LIN {X 0,Y 474.701,Z 198.658,A -85,B 0,C 180,E1 -7391.962,E2 -7391.962} C_VEL
LIN {X 0,Y 474.697,Z 198.664,A -85,B 0,C 180,E1 -7395.456,E2 -7395.456} C_VEL
LIN {X 0,Y 474.662,Z 198.657,A -85,B 0,C 180,E1 -7399.01,E2 -7399.01} C_VEL
LIN {X 0,Y 474.586,Z 198.681,A -85,B 0,C 180,E1 -7401.729,E2 -7401.729} C_VEL
LIN {X 0,Y 474.656,Z 198.662,A -85,B 0,C 180,E1 -7404.493,E2 -7404.493} C_VEL
LIN {X 0,Y 474.697,Z 198.662,A -85,B 0,C 180,E1 -7407.339,E2 -7407.339} C_VEL
LIN {X 0,Y 474.606,Z 198.671,A -85,B 0,C 180,E1 -7410.811,E2 -7410.811} C_VEL
LIN {X 0,Y 474.636,Z 198.675,A -85,B 0,C 180,E1 -7413.984,E2 -7413.984} C_VEL
LIN {X 0,Y 474.572,Z 198.677,A -85,B 0,C 180,E1 -7416.9,E2 -7416.9} C_VEL
LIN {X 0,Y 474.625,Z 198.675,A -85,B 0,C 180,E1 -7419.648,E2 -7419.648} C_VEL
LIN {X 0,Y 474.612,Z 198.673,A -85,B 0,C 180,E1 -7422.934,E2 -7422.934} C_VEL
LIN {X 0,Y 474.604,Z 198.679,A -85,B 0,C 180,E1 -7425.895,E2 -7425.895} C_VEL
LIN {X 0,Y 474.625,Z 198.671,A -85,B 0,C 180,E1 -7429.041,E2 -7429.041} C_VEL
LIN {X 0,Y 474.608,Z 198.678,A -85,B 0,C 180,E1 -7431.704,E2 -7431.704} C_VEL
LIN {X 0,Y 474.623,Z 198.668,A -85,B 0,C 180,E1 -7434.726,E2 -7434.726} C_VEL
LIN {X 0,Y 474.635,Z 198.669,A -85,B 0,C 180,E1 -7437.788,E2 -7437.788} C_VEL
LIN {X 0,Y 474.623,Z 198.677,A -85,B 0,C 180,E1 -7440.885,E2 -7440.885} C_VEL
LIN {X 0,Y 474.66,Z 198.672,A -85,B 0,C 180,E1 -7443.628,E2 -7443.628} C_VEL
LIN {X 0,Y 474.635,Z 198.669,A -85,B 0,C 180,E1 -7446.641,E2 -7446.641} C_VEL
LIN {X 0,Y 474.653,Z 198.661,A -85,B 0,C 180,E1 -7450.09,E2 -7450.09} C_VEL
LIN {X 0,Y 474.646,Z 198.663,A -85,B 0,C 180,E1 -7451.677,E2 -7451.677} C_VEL
LIN {X 0,Y 473.979,Z 198.754,A -85,B 0,C 180,E1 -7452.386,E2 -7452.386} C_VEL
LIN {X 0,Y 471.131,Z 199.113,A -85,B 0,C 180,E1 -7453.537,E2 -7453.537} C_VEL
LIN {X 0,Y 468.721,Z 199.413,A -85,B 0,C 180,E1 -7454.466,E2 -7454.466} C_VEL
LIN {X 0,Y 467.682,Z 199.532,A -85,B 0,C 180,E1 -7455.183,E2 -7455.183} C_VEL
LIN {X 0,Y 467.596,Z 199.539,A -85,B 0,C 180,E1 -7455.426,E2 -7455.426} C_VEL
LIN {X 0,Y 467.653,Z 199.547,A -85,B 0,C 180,E1 -7458.734,E2 -7458.734} C_VEL
LIN {X 0,Y 467.681,Z 199.542,A -85,B 0,C 180,E1 -7461.357,E2 -7461.357} C_VEL
LIN {X 0,Y 467.723,Z 199.527,A -85,B 0,C 180,E1 -7463.962,E2 -7463.962} C_VEL
LIN {X 0,Y 467.656,Z 199.646,A -85,B 0,C 180,E1 -7465.367,E2 -7465.367} C_VEL
LIN {X 0,Y 470.553,Z 208.926,A -85,B 0,C 180,E1 -7466.72,E2 -7466.72} C_VEL
LIN {X 0,Y 480.237,Z 229.746,A -85,B 0,C 180,E1 -7467.714,E2 -7467.714} C_VEL
LIN {X 0,Y 477.501,Z 414.726,A -85,B 0,C 180,E1 -7470.658,E2 -7470.658} C_VEL
LIN {X 0,Y 476.956,Z 430.924,A -85,B 0,C 180,E1 -7471.082,E2 -7471.082} C_VEL
LIN {X 0,Y 476.243,Z 446.299,A -85,B 0,C 180,E1 -7471.638,E2 -7471.638} C_VEL
LIN {X 0,Y 475.447,Z 461.115,A -85,B 0,C 180,E1 -7472.329,E2 -7472.329} C_VEL
LIN {X 0,Y 474.447,Z 475.812,A -85,B 0,C 180,E1 -7473.184,E2 -7473.184} C_VEL
LIN {X 0,Y 473.458,Z 489.457,A -85,B 0,C 180,E1 -7474.15,E2 -7474.15} C_VEL
LIN {X 0,Y 472.422,Z 503.502,A -85,B 0,C 180,E1 -7475.335,E2 -7475.335} C_VEL
LIN {X 0,Y 471.27,Z 516.574,A -85,B 0,C 180,E1 -7476.636,E2 -7476.636} C_VEL
LIN {X 0,Y 470.217,Z 529.445,A -85,B 0,C 180,E1 -7478.163,E2 -7478.163} C_VEL
LIN {X 0,Y 469.318,Z 540.358,A -85,B 0,C 180,E1 -7479.698,E2 -7479.698} C_VEL
LIN {X 0,Y 468.563,Z 549.76,A -85,B 0,C 180,E1 -7481.244,E2 -7481.244} C_VEL
LIN {X 0,Y 467.904,Z 558.942,A -85,B 0,C 180,E1 -7483.02,E2 -7483.02} C_VEL
LIN {X 0,Y 467.402,Z 566.666,A -85,B 0,C 180,E1 -7484.81,E2 -7484.81} C_VEL
LIN {X 0,Y 467.041,Z 572.995,A -85,B 0,C 180,E1 -7486.613,E2 -7486.613} C_VEL
LIN {X 0,Y 466.832,Z 578.273,A -85,B 0,C 180,E1 -7488.479,E2 -7488.479} C_VEL
LIN {X 0,Y 466.666,Z 582.208,A -85,B 0,C 180,E1 -7490.266,E2 -7490.266} C_VEL
LIN {X 0,Y 466.519,Z 585.068,A -85,B 0,C 180,E1 -7492.124,E2 -7492.124} C_VEL
LIN {X 0,Y 466.463,Z 586.873,A -85,B 0,C 180,E1 -7494.003,E2 -7494.003} C_VEL
LIN {X 0,Y 466.465,Z 587.555,A -85,B 0,C 180,E1 -7495.907,E2 -7495.907} C_VEL
LIN {X 0,Y 466.492,Z 587.024,A -85,B 0,C 180,E1 -7497.841,E2 -7497.841} C_VEL
LIN {X 0,Y 466.581,Z 585.307,A -85,B 0,C 180,E1 -7499.806,E2 -7499.806} C_VEL
LIN {X 0,Y 466.679,Z 582.29,A -85,B 0,C 180,E1 -7501.808,E2 -7501.808} C_VEL
LIN {X 0,Y 466.876,Z 577.769,A -85,B 0,C 180,E1 -7503.846,E2 -7503.846} C_VEL
LIN {X 0,Y 467.13,Z 572.464,A -85,B 0,C 180,E1 -7505.666,E2 -7505.666} C_VEL
LIN {X 0,Y 467.494,Z 565.604,A -85,B 0,C 180,E1 -7507.565,E2 -7507.565} C_VEL
LIN {X 0,Y 467.974,Z 557.8,A -85,B 0,C 180,E1 -7509.346,E2 -7509.346} C_VEL
LIN {X 0,Y 468.743,Z 547.515,A -85,B 0,C 180,E1 -7511.276,E2 -7511.276} C_VEL
LIN {X 0,Y 469.535,Z 537.645,A -85,B 0,C 180,E1 -7512.825,E2 -7512.825} C_VEL
LIN {X 0,Y 470.512,Z 526.433,A -85,B 0,C 180,E1 -7514.331,E2 -7514.331} C_VEL
LIN {X 0,Y 471.498,Z 514.718,A -85,B 0,C 180,E1 -7515.681,E2 -7515.681} C_VEL
LIN {X 0,Y 472.653,Z 500.994,A -85,B 0,C 180,E1 -7517.02,E2 -7517.02} C_VEL
LIN {X 0,Y 473.89,Z 485.591,A -85,B 0,C 180,E1 -7518.264,E2 -7518.264} C_VEL
LIN {X 0,Y 474.951,Z 470.284,A -85,B 0,C 180,E1 -7519.276,E2 -7519.276} C_VEL
LIN {X 0,Y 475.877,Z 454.74,A -85,B 0,C 180,E1 -7520.105,E2 -7520.105} C_VEL
LIN {X 0,Y 476.698,Z 438.378,A -85,B 0,C 180,E1 -7520.786,E2 -7520.786} C_VEL
LIN {X 0,Y 477.348,Z 421.885,A -85,B 0,C 180,E1 -7521.289,E2 -7521.289} C_VEL
LIN {X 0,Y 477.799,Z 404.177,A -85,B 0,C 180,E1 -7521.642,E2 -7521.642} C_VEL
LIN {X 0,Y 480.393,Z 230.17,A -85,B 0,C 180,E1 -7524.41,E2 -7524.41} C_VEL
LIN {X 0,Y 471.537,Z 211.431,A -85,B 0,C 180,E1 -7525.341,E2 -7525.341} C_VEL
LIN {X 0,Y 470.535,Z 209.235,A -85,B 0,C 180,E1 -7525.46,E2 -7525.46} C_VEL
LIN {X 0,Y 467.562,Z 199.56,A -85,B 0,C 180,E1 -7526.952,E2 -7526.952} C_VEL
LIN {X 0,Y 467.56,Z 199.557,A -85,B 0,C 180,E1 -7529.266,E2 -7529.266} C_VEL
LIN {X 0,Y 467.596,Z 199.554,A -85,B 0,C 180,E1 -7532.469,E2 -7532.469} C_VEL
LIN {X 0,Y 467.552,Z 199.556,A -85,B 0,C 180,E1 -7535.11,E2 -7535.11} C_VEL
LIN {X 0,Y 467.526,Z 199.554,A -85,B 0,C 180,E1 -7537.926,E2 -7537.926} C_VEL
LIN {X 0,Y 467.615,Z 199.547,A -85,B 0,C 180,E1 -7540.692,E2 -7540.692} C_VEL
LIN {X 0,Y 467.642,Z 199.541,A -85,B 0,C 180,E1 -7544.115,E2 -7544.115} C_VEL
LIN {X 0,Y 467.647,Z 199.538,A -85,B 0,C 180,E1 -7547.642,E2 -7547.642} C_VEL
LIN {X 0,Y 467.654,Z 199.547,A -85,B 0,C 180,E1 -7550.485,E2 -7550.485} C_VEL
LIN {X 0,Y 467.683,Z 199.537,A -85,B 0,C 180,E1 -7553.095,E2 -7553.095} C_VEL
LIN {X 0,Y 467.712,Z 199.536,A -85,B 0,C 180,E1 -7554.827,E2 -7554.827} C_VEL
LIN {X 0,Y 467.851,Z 199.517,A -85,B 0,C 180,E1 -7557.417,E2 -7557.417} C_VEL
LIN {X 0,Y 467.875,Z 199.518,A -85,B 0,C 180,E1 -7560,E2 -7560} C_VEL
LIN {X 0,Y 467.852,Z 199.518,A -85,B 0,C 180,E1 -7562.583,E2 -7562.583} C_VEL
LIN {X 0,Y 467.736,Z 199.534,A -85,B 0,C 180,E1 -7566.037,E2 -7566.037} C_VEL
LIN {X 0,Y 467.675,Z 199.54,A -85,B 0,C 180,E1 -7568.643,E2 -7568.643} C_VEL
LIN {X 0,Y 467.649,Z 199.548,A -85,B 0,C 180,E1 -7572.146,E2 -7572.146} C_VEL
LIN {X 0,Y 467.632,Z 199.549,A -85,B 0,C 180,E1 -7575.695,E2 -7575.695} C_VEL
LIN {X 0,Y 467.611,Z 199.545,A -85,B 0,C 180,E1 -7578.765,E2 -7578.765} C_VEL
LIN {X 0,Y 467.574,Z 199.554,A -85,B 0,C 180,E1 -7581.269,E2 -7581.269} C_VEL
LIN {X 0,Y 467.567,Z 199.555,A -85,B 0,C 180,E1 -7583.943,E2 -7583.943} C_VEL
LIN {X 0,Y 467.621,Z 199.544,A -85,B 0,C 180,E1 -7586.8,E2 -7586.8} C_VEL
LIN {X 0,Y 467.548,Z 199.561,A -85,B 0,C 180,E1 -7589.738,E2 -7589.738} C_VEL
LIN {X 0,Y 467.578,Z 199.554,A -85,B 0,C 180,E1 -7592.759,E2 -7592.759} C_VEL
LIN {X 0,Y 467.548,Z 199.559,A -85,B 0,C 180,E1 -7595.89,E2 -7595.89} C_VEL
LIN {X 0,Y 467.577,Z 199.56,A -85,B 0,C 180,E1 -7599.145,E2 -7599.145} C_VEL
LIN {X 0,Y 467.581,Z 199.555,A -85,B 0,C 180,E1 -7602.567,E2 -7602.567} C_VEL
LIN {X 0,Y 467.565,Z 199.562,A -85,B 0,C 180,E1 -7605.054,E2 -7605.054} C_VEL
LIN {X 0,Y 467.584,Z 199.557,A -85,B 0,C 180,E1 -7607.44,E2 -7607.44} C_VEL
LIN {X 0,Y 467.578,Z 199.556,A -85,B 0,C 180,E1 -7610.856,E2 -7610.856} C_VEL
LIN {X 0,Y 467.555,Z 199.558,A -85,B 0,C 180,E1 -7614.261,E2 -7614.261} C_VEL
LIN {X 0,Y 467.623,Z 199.676,A -85,B 0,C 180,E1 -7616.717,E2 -7616.717} C_VEL
LIN {X 0,Y 473.655,Z 219.02,A -85,B 0,C 180,E1 -7619.383,E2 -7619.383} C_VEL
LIN {X 0,Y 475.73,Z 226.359,A -85,B 0,C 180,E1 -7620.338,E2 -7620.338} C_VEL
LIN {X 0,Y 475.601,Z 231.753,A -85,B 0,C 180,E1 -7620.923,E2 -7620.923} C_VEL
LIN {X 0,Y 480.058,Z 257.266,A -85,B 0,C 180,E1 -7621.669,E2 -7621.669} C_VEL
LIN {X 0,Y 478.155,Z 385.84,A -85,B 0,C 180,E1 -7623.713,E2 -7623.713} C_VEL
LIN {X 0,Y 477.384,Z 438.968,A -85,B 0,C 180,E1 -7624.572,E2 -7624.572} C_VEL
LIN {X 0,Y 476.72,Z 455.187,A -85,B 0,C 180,E1 -7624.981,E2 -7624.981} C_VEL
LIN {X 0,Y 475.931,Z 471.769,A -85,B 0,C 180,E1 -7625.577,E2 -7625.577} C_VEL
LIN {X 0,Y 475.084,Z 485.876,A -85,B 0,C 180,E1 -7626.228,E2 -7626.228} C_VEL
LIN {X 0,Y 474.059,Z 501.348,A -85,B 0,C 180,E1 -7627.124,E2 -7627.124} C_VEL
LIN {X 0,Y 472.982,Z 514.94,A -85,B 0,C 180,E1 -7628.079,E2 -7628.079} C_VEL
LIN {X 0,Y 471.805,Z 529.315,A -85,B 0,C 180,E1 -7629.282,E2 -7629.282} C_VEL
LIN {X 0,Y 470.709,Z 542.794,A -85,B 0,C 180,E1 -7630.625,E2 -7630.625} C_VEL
LIN {X 0,Y 469.852,Z 553.86,A -85,B 0,C 180,E1 -7631.919,E2 -7631.919} C_VEL
LIN {X 0,Y 468.922,Z 565.152,A -85,B 0,C 180,E1 -7633.456,E2 -7633.456} C_VEL
LIN {X 0,Y 468.276,Z 574.848,A -85,B 0,C 180,E1 -7634.996,E2 -7634.996} C_VEL
LIN {X 0,Y 467.651,Z 584.267,A -85,B 0,C 180,E1 -7636.752,E2 -7636.752} C_VEL
LIN {X 0,Y 467.337,Z 591.16,A -85,B 0,C 180,E1 -7638.287,E2 -7638.287} C_VEL
LIN {X 0,Y 466.969,Z 597.843,A -85,B 0,C 180,E1 -7640.034,E2 -7640.034} C_VEL
LIN {X 0,Y 466.79,Z 603.262,A -85,B 0,C 180,E1 -7641.777,E2 -7641.777} C_VEL
LIN {X 0,Y 466.748,Z 607.738,A -85,B 0,C 180,E1 -7643.607,E2 -7643.607} C_VEL
LIN {X 0,Y 466.599,Z 611.426,A -85,B 0,C 180,E1 -7645.681,E2 -7645.681} C_VEL
LIN {X 0,Y 466.651,Z 613.384,A -85,B 0,C 180,E1 -7647.411,E2 -7647.411} C_VEL
LIN {X 0,Y 466.615,Z 614.358,A -85,B 0,C 180,E1 -7649.137,E2 -7649.137} C_VEL
LIN {X 0,Y 466.615,Z 614.364,A -85,B 0,C 180,E1 -7650.863,E2 -7650.863} C_VEL
LIN {X 0,Y 466.651,Z 613.402,A -85,B 0,C 180,E1 -7652.59,E2 -7652.59} C_VEL
LIN {X 0,Y 466.599,Z 611.458,A -85,B 0,C 180,E1 -7654.319,E2 -7654.319} C_VEL
LIN {X 0,Y 466.749,Z 607.791,A -85,B 0,C 180,E1 -7656.393,E2 -7656.393} C_VEL
LIN {X 0,Y 466.791,Z 603.33,A -85,B 0,C 180,E1 -7658.223,E2 -7658.223} C_VEL
LIN {X 0,Y 466.97,Z 597.926,A -85,B 0,C 180,E1 -7659.967,E2 -7659.967} C_VEL
LIN {X 0,Y 467.341,Z 591.258,A -85,B 0,C 180,E1 -7661.714,E2 -7661.714} C_VEL
LIN {X 0,Y 467.737,Z 583.265,A -85,B 0,C 180,E1 -7663.468,E2 -7663.468} C_VEL
LIN {X 0,Y 468.437,Z 573.726,A -85,B 0,C 180,E1 -7665.222,E2 -7665.222} C_VEL
LIN {X 0,Y 469.225,Z 562.294,A -85,B 0,C 180,E1 -7666.982,E2 -7666.982} C_VEL
LIN {X 0,Y 470.17,Z 550.41,A -85,B 0,C 180,E1 -7668.52,E2 -7668.52} C_VEL
LIN {X 0,Y 471.132,Z 538.262,A -85,B 0,C 180,E1 -7669.864,E2 -7669.864} C_VEL
LIN {X 0,Y 472.226,Z 524.526,A -85,B 0,C 180,E1 -7671.156,E2 -7671.156} C_VEL
LIN {X 0,Y 473.297,Z 510.729,A -85,B 0,C 180,E1 -7672.25,E2 -7672.25} C_VEL
LIN {X 0,Y 474.486,Z 494.972,A -85,B 0,C 180,E1 -7673.273,E2 -7673.273} C_VEL
LIN {X 0,Y 475.503,Z 479.167,A -85,B 0,C 180,E1 -7674.098,E2 -7674.098} C_VEL
LIN {X 0,Y 476.37,Z 463.217,A -85,B 0,C 180,E1 -7674.748,E2 -7674.748} C_VEL
LIN {X 0,Y 477.018,Z 447.128,A -85,B 0,C 180,E1 -7675.236,E2 -7675.236} C_VEL
LIN {X 0,Y 477.593,Z 430.192,A -85,B 0,C 180,E1 -7675.571,E2 -7675.571} C_VEL
LIN {X 0,Y 479.963,Z 257.006,A -85,B 0,C 180,E1 -7678.31,E2 -7678.31} C_VEL
LIN {X 0,Y 475.587,Z 232.12,A -85,B 0,C 180,E1 -7679.04,E2 -7679.04} C_VEL
LIN {X 0,Y 475.709,Z 226.306,A -85,B 0,C 180,E1 -7679.667,E2 -7679.667} C_VEL
LIN {X 0,Y 470.359,Z 208.522,A -85,B 0,C 180,E1 -7682.012,E2 -7682.012} C_VEL
LIN {X 0,Y 467.612,Z 199.535,A -85,B 0,C 180,E1 -7683.269,E2 -7683.269} C_VEL
LIN {X 0,Y 467.549,Z 199.558,A -85,B 0,C 180,E1 -7685.89,E2 -7685.89} C_VEL
LIN {X 0,Y 467.568,Z 199.557,A -85,B 0,C 180,E1 -7689.146,E2 -7689.146} C_VEL
LIN {X 0,Y 467.57,Z 199.557,A -85,B 0,C 180,E1 -7691.403,E2 -7691.403} C_VEL
LIN {X 0,Y 467.562,Z 199.554,A -85,B 0,C 180,E1 -7695.052,E2 -7695.052} C_VEL
LIN {X 0,Y 467.57,Z 199.555,A -85,B 0,C 180,E1 -7698.597,E2 -7698.597} C_VEL
LIN {X 0,Y 467.561,Z 199.554,A -85,B 0,C 180,E1 -7701.955,E2 -7701.955} C_VEL
LIN {X 0,Y 467.555,Z 199.558,A -85,B 0,C 180,E1 -7705.167,E2 -7705.167} C_VEL
LIN {X 0,Y 467.579,Z 199.545,A -85,B 0,C 180,E1 -7708.26,E2 -7708.26} C_VEL
LIN {X 0,Y 467.572,Z 199.554,A -85,B 0,C 180,E1 -7711.25,E2 -7711.25} C_VEL
LIN {X 0,Y 467.594,Z 199.539,A -85,B 0,C 180,E1 -7714.159,E2 -7714.159} C_VEL
LIN {X 0,Y 467.572,Z 199.556,A -85,B 0,C 180,E1 -7716.996,E2 -7716.996} C_VEL
LIN {X 0,Y 467.618,Z 199.539,A -85,B 0,C 180,E1 -7719.777,E2 -7719.777} C_VEL
LIN {X 0,Y 467.592,Z 199.546,A -85,B 0,C 180,E1 -7722.506,E2 -7722.506} C_VEL
LIN {X 0,Y 467.602,Z 199.547,A -85,B 0,C 180,E1 -7725.196,E2 -7725.196} C_VEL
LIN {X 0,Y 467.653,Z 199.53,A -85,B 0,C 180,E1 -7727.855,E2 -7727.855} C_VEL
LIN {X 0,Y 467.667,Z 199.538,A -85,B 0,C 180,E1 -7731.357,E2 -7731.357} C_VEL
LIN {X 0,Y 467.73,Z 199.534,A -85,B 0,C 180,E1 -7733.962,E2 -7733.962} C_VEL
LIN {X 0,Y 467.854,Z 199.495,A -85,B 0,C 180,E1 -7737.417,E2 -7737.417} C_VEL
LIN {X 0,Y 467.878,Z 199.511,A -85,B 0,C 180,E1 -7740,E2 -7740} C_VEL
LIN {X 0,Y 467.855,Z 199.517,A -85,B 0,C 180,E1 -7742.583,E2 -7742.583} C_VEL
LIN {X 0,Y 467.739,Z 199.524,A -85,B 0,C 180,E1 -7746.037,E2 -7746.037} C_VEL
LIN {X 0,Y 467.677,Z 199.539,A -85,B 0,C 180,E1 -7748.643,E2 -7748.643} C_VEL
LIN {X 0,Y 467.653,Z 199.535,A -85,B 0,C 180,E1 -7752.145,E2 -7752.145} C_VEL
LIN {X 0,Y 467.636,Z 199.546,A -85,B 0,C 180,E1 -7755.695,E2 -7755.695} C_VEL
LIN {X 0,Y 467.614,Z 199.534,A -85,B 0,C 180,E1 -7758.765,E2 -7758.765} C_VEL
LIN {X 0,Y 467.578,Z 199.549,A -85,B 0,C 180,E1 -7761.268,E2 -7761.268} C_VEL
LIN {X 0,Y 467.571,Z 199.55,A -85,B 0,C 180,E1 -7763.943,E2 -7763.943} C_VEL
LIN {X 0,Y 467.614,Z 199.541,A -85,B 0,C 180,E1 -7766.8,E2 -7766.8} C_VEL
LIN {X 0,Y 467.584,Z 199.555,A -85,B 0,C 180,E1 -7769.736,E2 -7769.736} C_VEL
LIN {X 0,Y 467.581,Z 199.543,A -85,B 0,C 180,E1 -7772.758,E2 -7772.758} C_VEL
LIN {X 0,Y 467.554,Z 199.556,A -85,B 0,C 180,E1 -7775.889,E2 -7775.889} C_VEL
LIN {X 0,Y 467.579,Z 199.545,A -85,B 0,C 180,E1 -7779.145,E2 -7779.145} C_VEL
LIN {X 0,Y 467.584,Z 199.547,A -85,B 0,C 180,E1 -7782.567,E2 -7782.567} C_VEL
LIN {X 0,Y 467.563,Z 199.55,A -85,B 0,C 180,E1 -7785.053,E2 -7785.053} C_VEL
LIN {X 0,Y 467.587,Z 199.554,A -85,B 0,C 180,E1 -7787.44,E2 -7787.44} C_VEL
LIN {X 0,Y 467.558,Z 199.553,A -85,B 0,C 180,E1 -7790.853,E2 -7790.853} C_VEL
LIN {X 0,Y 467.558,Z 199.547,A -85,B 0,C 180,E1 -7794.261,E2 -7794.261} C_VEL
LIN {X 0,Y 467.581,Z 199.554,A -85,B 0,C 180,E1 -7797.321,E2 -7797.321} C_VEL
LIN {X 0,Y 467.569,Z 199.554,A -85,B 0,C 180,E1 -7800.667,E2 -7800.667} C_VEL
LIN {X 0,Y 467.616,Z 199.547,A -85,B 0,C 180,E1 -7803.2,E2 -7803.2} C_VEL
LIN {X 0,Y 467.592,Z 199.545,A -85,B 0,C 180,E1 -7806.468,E2 -7806.468} C_VEL
LIN {X 0,Y 467.622,Z 199.538,A -85,B 0,C 180,E1 -7809.777,E2 -7809.777} C_VEL
LIN {X 0,Y 467.597,Z 199.545,A -85,B 0,C 180,E1 -7812.506,E2 -7812.506} C_VEL
LIN {X 0,Y 467.605,Z 199.541,A -85,B 0,C 180,E1 -7815.196,E2 -7815.196} C_VEL
LIN {X 0,Y 467.596,Z 199.539,A -85,B 0,C 180,E1 -7815.426,E2 -7815.426} C_VEL
LIN {X 0,Y 466.926,Z 199.621,A -85,B 0,C 180,E1 -7816.145,E2 -7816.145} C_VEL
LIN {X 0,Y 464.083,Z 199.985,A -85,B 0,C 180,E1 -7817.314,E2 -7817.314} C_VEL
LIN {X 0,Y 461.684,Z 200.288,A -85,B 0,C 180,E1 -7818.256,E2 -7818.256} C_VEL
LIN {X 0,Y 460.658,Z 200.416,A -85,B 0,C 180,E1 -7818.983,E2 -7818.983} C_VEL
LIN {X 0,Y 460.576,Z 200.425,A -85,B 0,C 180,E1 -7819.23,E2 -7819.23} C_VEL
LIN {X 0,Y 460.669,Z 200.411,A -85,B 0,C 180,E1 -7822.587,E2 -7822.587} C_VEL
LIN {X 0,Y 460.655,Z 200.475,A -85,B 0,C 180,E1 -7824.94,E2 -7824.94} C_VEL
LIN {X 0,Y 463.309,Z 209.246,A -85,B 0,C 180,E1 -7826.227,E2 -7826.227} C_VEL
LIN {X 0,Y 470.395,Z 224.099,A -85,B 0,C 180,E1 -7826.973,E2 -7826.973} C_VEL
LIN {X 0,Y 473.966,Z 231.809,A -85,B 0,C 180,E1 -7827.344,E2 -7827.344} C_VEL
LIN {X 0,Y 471.072,Z 414.547,A -85,B 0,C 180,E1 -7830.288,E2 -7830.288} C_VEL
LIN {X 0,Y 470.511,Z 430.619,A -85,B 0,C 180,E1 -7830.708,E2 -7830.708} C_VEL
LIN {X 0,Y 469.744,Z 446.47,A -85,B 0,C 180,E1 -7831.286,E2 -7831.286} C_VEL
LIN {X 0,Y 468.982,Z 460.305,A -85,B 0,C 180,E1 -7831.932,E2 -7831.932} C_VEL
LIN {X 0,Y 467.809,Z 476.864,A -85,B 0,C 180,E1 -7832.906,E2 -7832.906} C_VEL
LIN {X 0,Y 466.677,Z 491.742,A -85,B 0,C 180,E1 -7833.994,E2 -7833.994} C_VEL
LIN {X 0,Y 465.566,Z 505.446,A -85,B 0,C 180,E1 -7835.196,E2 -7835.196} C_VEL
LIN {X 0,Y 464.375,Z 518.236,A -85,B 0,C 180,E1 -7836.517,E2 -7836.517} C_VEL
LIN {X 0,Y 463.266,Z 530.89,A -85,B 0,C 180,E1 -7838.066,E2 -7838.066} C_VEL
LIN {X 0,Y 462.337,Z 541.697,A -85,B 0,C 180,E1 -7839.625,E2 -7839.625} C_VEL
LIN {X 0,Y 461.458,Z 552.148,A -85,B 0,C 180,E1 -7841.419,E2 -7841.419} C_VEL
LIN {X 0,Y 460.771,Z 560.953,A -85,B 0,C 180,E1 -7843.225,E2 -7843.225} C_VEL
LIN {X 0,Y 460.282,Z 568.34,A -85,B 0,C 180,E1 -7845.044,E2 -7845.044} C_VEL
LIN {X 0,Y 459.953,Z 574.477,A -85,B 0,C 180,E1 -7846.876,E2 -7846.876} C_VEL
LIN {X 0,Y 459.733,Z 579.339,A -85,B 0,C 180,E1 -7848.725,E2 -7848.725} C_VEL
LIN {X 0,Y 459.539,Z 583.111,A -85,B 0,C 180,E1 -7850.594,E2 -7850.594} C_VEL
LIN {X 0,Y 459.405,Z 585.806,A -85,B 0,C 180,E1 -7852.485,E2 -7852.485} C_VEL
LIN {X 0,Y 459.364,Z 587.309,A -85,B 0,C 180,E1 -7854.398,E2 -7854.398} C_VEL
LIN {X 0,Y 459.377,Z 587.734,A -85,B 0,C 180,E1 -7856.338,E2 -7856.338} C_VEL
LIN {X 0,Y 459.411,Z 586.996,A -85,B 0,C 180,E1 -7858.309,E2 -7858.309} C_VEL
LIN {X 0,Y 459.494,Z 584.949,A -85,B 0,C 180,E1 -7860.313,E2 -7860.313} C_VEL
LIN {X 0,Y 459.646,Z 581.583,A -85,B 0,C 180,E1 -7862.353,E2 -7862.353} C_VEL
LIN {X 0,Y 459.884,Z 576.747,A -85,B 0,C 180,E1 -7864.432,E2 -7864.432} C_VEL
LIN {X 0,Y 460.141,Z 571.404,A -85,B 0,C 180,E1 -7866.215,E2 -7866.215} C_VEL
LIN {X 0,Y 460.574,Z 564.098,A -85,B 0,C 180,E1 -7868.169,E2 -7868.169} C_VEL
LIN {X 0,Y 461.206,Z 555.292,A -85,B 0,C 180,E1 -7870.096,E2 -7870.096} C_VEL
LIN {X 0,Y 461.998,Z 545.931,A -85,B 0,C 180,E1 -7871.807,E2 -7871.807} C_VEL
LIN {X 0,Y 462.872,Z 535.742,A -85,B 0,C 180,E1 -7873.395,E2 -7873.395} C_VEL
LIN {X 0,Y 463.949,Z 524.199,A -85,B 0,C 180,E1 -7874.916,E2 -7874.916} C_VEL
LIN {X 0,Y 465.058,Z 511.855,A -85,B 0,C 180,E1 -7876.298,E2 -7876.298} C_VEL
LIN {X 0,Y 466.213,Z 497.981,A -85,B 0,C 180,E1 -7877.616,E2 -7877.616} C_VEL
LIN {X 0,Y 467.414,Z 483.724,A -85,B 0,C 180,E1 -7878.745,E2 -7878.745} C_VEL
LIN {X 0,Y 468.469,Z 469.786,A -85,B 0,C 180,E1 -7879.665,E2 -7879.665} C_VEL
LIN {X 0,Y 469.488,Z 453.715,A -85,B 0,C 180,E1 -7880.52,E2 -7880.52} C_VEL
LIN {X 0,Y 470.295,Z 437.805,A -85,B 0,C 180,E1 -7881.179,E2 -7881.179} C_VEL
LIN {X 0,Y 471.011,Z 421.355,A -85,B 0,C 180,E1 -7881.675,E2 -7881.675} C_VEL
LIN {X 0,Y 471.426,Z 404.144,A -85,B 0,C 180,E1 -7882.021,E2 -7882.021} C_VEL
LIN {X 0,Y 474.192,Z 232.29,A -85,B 0,C 180,E1 -7884.79,E2 -7884.79} C_VEL
LIN {X 0,Y 464.605,Z 212.097,A -85,B 0,C 180,E1 -7885.828,E2 -7885.828} C_VEL
LIN {X 0,Y 463.367,Z 209.366,A -85,B 0,C 180,E1 -7885.993,E2 -7885.993} C_VEL
LIN {X 0,Y 460.528,Z 200.433,A -85,B 0,C 180,E1 -7887.397,E2 -7887.397} C_VEL
LIN {X 0,Y 460.519,Z 200.434,A -85,B 0,C 180,E1 -7890.768,E2 -7890.768} C_VEL
LIN {X 0,Y 460.511,Z 200.434,A -85,B 0,C 180,E1 -7893.732,E2 -7893.732} C_VEL
LIN {X 0,Y 460.536,Z 200.434,A -85,B 0,C 180,E1 -7896.624,E2 -7896.624} C_VEL
LIN {X 0,Y 460.543,Z 200.431,A -85,B 0,C 180,E1 -7899.452,E2 -7899.452} C_VEL
LIN {X 0,Y 460.542,Z 200.43,A -85,B 0,C 180,E1 -7902.23,E2 -7902.23} C_VEL
LIN {X 0,Y 460.557,Z 200.426,A -85,B 0,C 180,E1 -7904.965,E2 -7904.965} C_VEL
LIN {X 0,Y 460.603,Z 200.417,A -85,B 0,C 180,E1 -7908.559,E2 -7908.559} C_VEL
LIN {X 0,Y 460.613,Z 200.419,A -85,B 0,C 180,E1 -7911.224,E2 -7911.224} C_VEL
LIN {X 0,Y 460.691,Z 200.408,A -85,B 0,C 180,E1 -7913.87,E2 -7913.87} C_VEL
LIN {X 0,Y 460.792,Z 200.396,A -85,B 0,C 180,E1 -7917.377,E2 -7917.377} C_VEL
LIN {X 0,Y 460.845,Z 200.394,A -85,B 0,C 180,E1 -7920,E2 -7920} C_VEL
LIN {X 0,Y 460.793,Z 200.397,A -85,B 0,C 180,E1 -7922.623,E2 -7922.623} C_VEL
LIN {X 0,Y 460.702,Z 200.411,A -85,B 0,C 180,E1 -7926.13,E2 -7926.13} C_VEL
LIN {X 0,Y 460.622,Z 200.418,A -85,B 0,C 180,E1 -7928.776,E2 -7928.776} C_VEL
LIN {X 0,Y 460.607,Z 200.422,A -85,B 0,C 180,E1 -7932.445,E2 -7932.445} C_VEL
LIN {X 0,Y 460.593,Z 200.424,A -85,B 0,C 180,E1 -7935.998,E2 -7935.998} C_VEL
LIN {X 0,Y 460.564,Z 200.423,A -85,B 0,C 180,E1 -7938.902,E2 -7938.902} C_VEL
LIN {X 0,Y 460.51,Z 200.435,A -85,B 0,C 180,E1 -7941.486,E2 -7941.486} C_VEL
LIN {X 0,Y 460.536,Z 200.428,A -85,B 0,C 180,E1 -7944.332,E2 -7944.332} C_VEL
LIN {X 0,Y 460.578,Z 200.424,A -85,B 0,C 180,E1 -7947.243,E2 -7947.243} C_VEL
LIN {X 0,Y 460.505,Z 200.434,A -85,B 0,C 180,E1 -7950.24,E2 -7950.24} C_VEL
LIN {X 0,Y 460.523,Z 200.436,A -85,B 0,C 180,E1 -7953.325,E2 -7953.325} C_VEL
LIN {X 0,Y 460.471,Z 200.439,A -85,B 0,C 180,E1 -7956.53,E2 -7956.53} C_VEL
LIN {X 0,Y 460.527,Z 200.434,A -85,B 0,C 180,E1 -7959.863,E2 -7959.863} C_VEL
LIN {X 0,Y 460.508,Z 200.44,A -85,B 0,C 180,E1 -7962.901,E2 -7962.901} C_VEL
LIN {X 0,Y 460.506,Z 200.437,A -85,B 0,C 180,E1 -7965.831,E2 -7965.831} C_VEL
LIN {X 0,Y 460.526,Z 200.435,A -85,B 0,C 180,E1 -7968.989,E2 -7968.989} C_VEL
LIN {X 0,Y 460.522,Z 200.435,A -85,B 0,C 180,E1 -7971.267,E2 -7971.267} C_VEL
LIN {X 0,Y 460.506,Z 200.437,A -85,B 0,C 180,E1 -7974.555,E2 -7974.555} C_VEL
LIN {X 0,Y 460.575,Z 200.515,A -85,B 0,C 180,E1 -7976.247,E2 -7976.247} C_VEL
LIN {X 0,Y 466.904,Z 220.645,A -85,B 0,C 180,E1 -7979.09,E2 -7979.09} C_VEL
LIN {X 0,Y 469.168,Z 228.639,A -85,B 0,C 180,E1 -7980.153,E2 -7980.153} C_VEL
LIN {X 0,Y 469.148,Z 231.612,A -85,B 0,C 180,E1 -7980.485,E2 -7980.485} C_VEL
LIN {X 0,Y 473.829,Z 258.396,A -85,B 0,C 180,E1 -7981.278,E2 -7981.278} C_VEL
LIN {X 0,Y 472.073,Z 367.989,A -85,B 0,C 180,E1 -7983.043,E2 -7983.043} C_VEL
LIN {X 0,Y 470.982,Z 439.154,A -85,B 0,C 180,E1 -7984.207,E2 -7984.207} C_VEL
LIN {X 0,Y 470.254,Z 455.927,A -85,B 0,C 180,E1 -7984.643,E2 -7984.643} C_VEL
LIN {X 0,Y 469.454,Z 471.57,A -85,B 0,C 180,E1 -7985.218,E2 -7985.218} C_VEL
LIN {X 0,Y 468.538,Z 485.67,A -85,B 0,C 180,E1 -7985.875,E2 -7985.875} C_VEL
LIN {X 0,Y 467.506,Z 500.567,A -85,B 0,C 180,E1 -7986.747,E2 -7986.747} C_VEL
LIN {X 0,Y 466.318,Z 514.722,A -85,B 0,C 180,E1 -7987.75,E2 -7987.75} C_VEL
LIN {X 0,Y 465.094,Z 529.093,A -85,B 0,C 180,E1 -7988.969,E2 -7988.969} C_VEL
LIN {X 0,Y 464.022,Z 541.237,A -85,B 0,C 180,E1 -7990.179,E2 -7990.179} C_VEL
LIN {X 0,Y 463.004,Z 553.639,A -85,B 0,C 180,E1 -7991.642,E2 -7991.642} C_VEL
LIN {X 0,Y 462.009,Z 564.929,A -85,B 0,C 180,E1 -7993.201,E2 -7993.201} C_VEL
LIN {X 0,Y 461.336,Z 574.626,A -85,B 0,C 180,E1 -7994.765,E2 -7994.765} C_VEL
LIN {X 0,Y 460.646,Z 584.047,A -85,B 0,C 180,E1 -7996.546,E2 -7996.546} C_VEL
LIN {X 0,Y 460.166,Z 592.774,A -85,B 0,C 180,E1 -7998.548,E2 -7998.548} C_VEL
LIN {X 0,Y 459.775,Z 600.512,A -85,B 0,C 180,E1 -8000.764,E2 -8000.764} C_VEL
LIN {X 0,Y 459.647,Z 606.401,A -85,B 0,C 180,E1 -8002.974,E2 -8002.974} C_VEL
LIN {X 0,Y 459.578,Z 609.849,A -85,B 0,C 180,E1 -8004.736,E2 -8004.736} C_VEL
LIN {X 0,Y 459.53,Z 612.355,A -85,B 0,C 180,E1 -8006.493,E2 -8006.493} C_VEL
LIN {X 0,Y 459.537,Z 613.773,A -85,B 0,C 180,E1 -8008.247,E2 -8008.247} C_VEL
LIN {X 0,Y 459.525,Z 614.311,A -85,B 0,C 180,E1 -8010,E2 -8010} C_VEL
LIN {X 0,Y 459.537,Z 613.787,A -85,B 0,C 180,E1 -8011.753,E2 -8011.753} C_VEL
LIN {X 0,Y 459.53,Z 612.382,A -85,B 0,C 180,E1 -8013.507,E2 -8013.507} C_VEL
LIN {X 0,Y 459.578,Z 609.892,A -85,B 0,C 180,E1 -8015.265,E2 -8015.265} C_VEL
LIN {X 0,Y 459.648,Z 606.461,A -85,B 0,C 180,E1 -8017.026,E2 -8017.026} C_VEL
LIN {X 0,Y 459.782,Z 600.591,A -85,B 0,C 180,E1 -8019.236,E2 -8019.236} C_VEL
LIN {X 0,Y 460.172,Z 592.867,A -85,B 0,C 180,E1 -8021.452,E2 -8021.452} C_VEL
LIN {X 0,Y 460.648,Z 584.155,A -85,B 0,C 180,E1 -8023.454,E2 -8023.454} C_VEL
LIN {X 0,Y 461.36,Z 574.747,A -85,B 0,C 180,E1 -8025.235,E2 -8025.235} C_VEL
LIN {X 0,Y 462.071,Z 565.053,A -85,B 0,C 180,E1 -8026.797,E2 -8026.797} C_VEL
LIN {X 0,Y 463.008,Z 553.755,A -85,B 0,C 180,E1 -8028.359,E2 -8028.359} C_VEL
LIN {X 0,Y 464.066,Z 541.342,A -85,B 0,C 180,E1 -8029.82,E2 -8029.82} C_VEL
LIN {X 0,Y 465.212,Z 527.998,A -85,B 0,C 180,E1 -8031.142,E2 -8031.142} C_VEL
LIN {X 0,Y 466.32,Z 514.76,A -85,B 0,C 180,E1 -8032.251,E2 -8032.251} C_VEL
LIN {X 0,Y 467.497,Z 500.499,A -85,B 0,C 180,E1 -8033.256,E2 -8033.256} C_VEL
LIN {X 0,Y 468.552,Z 485.569,A -85,B 0,C 180,E1 -8034.125,E2 -8034.125} C_VEL
LIN {X 0,Y 469.517,Z 470.032,A -85,B 0,C 180,E1 -8034.838,E2 -8034.838} C_VEL
LIN {X 0,Y 470.27,Z 453.573,A -85,B 0,C 180,E1 -8035.416,E2 -8035.416} C_VEL
LIN {X 0,Y 470.954,Z 436.774,A -85,B 0,C 180,E1 -8035.819,E2 -8035.819} C_VEL
LIN {X 0,Y 473.743,Z 259.378,A -85,B 0,C 180,E1 -8038.667,E2 -8038.667} C_VEL
LIN {X 0,Y 469.08,Z 232.203,A -85,B 0,C 180,E1 -8039.446,E2 -8039.446} C_VEL
LIN {X 0,Y 469.044,Z 228.304,A -85,B 0,C 180,E1 -8039.881,E2 -8039.881} C_VEL
LIN {X 0,Y 463.548,Z 209.982,A -85,B 0,C 180,E1 -8042.338,E2 -8042.338} C_VEL
LIN {X 0,Y 460.544,Z 200.421,A -85,B 0,C 180,E1 -8043.717,E2 -8043.717} C_VEL
LIN {X 0,Y 460.47,Z 200.442,A -85,B 0,C 180,E1 -8046.53,E2 -8046.53} C_VEL
LIN {X 0,Y 460.518,Z 200.428,A -85,B 0,C 180,E1 -8049.863,E2 -8049.863} C_VEL
LIN {X 0,Y 460.489,Z 200.434,A -85,B 0,C 180,E1 -8052.897,E2 -8052.897} C_VEL
LIN {X 0,Y 460.502,Z 200.428,A -85,B 0,C 180,E1 -8055.831,E2 -8055.831} C_VEL
LIN {X 0,Y 460.524,Z 200.428,A -85,B 0,C 180,E1 -8058.988,E2 -8058.988} C_VEL
LIN {X 0,Y 460.513,Z 200.436,A -85,B 0,C 180,E1 -8061.266,E2 -8061.266} C_VEL
LIN {X 0,Y 460.505,Z 200.428,A -85,B 0,C 180,E1 -8064.554,E2 -8064.554} C_VEL
LIN {X 0,Y 460.527,Z 200.423,A -85,B 0,C 180,E1 -8067.715,E2 -8067.715} C_VEL
LIN {X 0,Y 460.535,Z 200.434,A -85,B 0,C 180,E1 -8070.769,E2 -8070.769} C_VEL
LIN {X 0,Y 460.552,Z 200.415,A -85,B 0,C 180,E1 -8073.734,E2 -8073.734} C_VEL
LIN {X 0,Y 460.541,Z 200.432,A -85,B 0,C 180,E1 -8076.624,E2 -8076.624} C_VEL
LIN {X 0,Y 460.547,Z 200.419,A -85,B 0,C 180,E1 -8079.453,E2 -8079.453} C_VEL
LIN {X 0,Y 460.544,Z 200.42,A -85,B 0,C 180,E1 -8082.23,E2 -8082.23} C_VEL
LIN {X 0,Y 460.561,Z 200.426,A -85,B 0,C 180,E1 -8084.965,E2 -8084.965} C_VEL
LIN {X 0,Y 460.607,Z 200.405,A -85,B 0,C 180,E1 -8088.559,E2 -8088.559} C_VEL
LIN {X 0,Y 460.617,Z 200.416,A -85,B 0,C 180,E1 -8091.224,E2 -8091.224} C_VEL
LIN {X 0,Y 460.695,Z 200.409,A -85,B 0,C 180,E1 -8093.87,E2 -8093.87} C_VEL
LIN {X 0,Y 460.795,Z 200.373,A -85,B 0,C 180,E1 -8097.377,E2 -8097.377} C_VEL
LIN {X 0,Y 460.848,Z 200.387,A -85,B 0,C 180,E1 -8100,E2 -8100} C_VEL
LIN {X 0,Y 460.796,Z 200.396,A -85,B 0,C 180,E1 -8102.623,E2 -8102.623} C_VEL
LIN {X 0,Y 460.705,Z 200.401,A -85,B 0,C 180,E1 -8106.13,E2 -8106.13} C_VEL
LIN {X 0,Y 460.624,Z 200.417,A -85,B 0,C 180,E1 -8108.776,E2 -8108.776} C_VEL
LIN {X 0,Y 460.611,Z 200.414,A -85,B 0,C 180,E1 -8112.445,E2 -8112.445} C_VEL
LIN {X 0,Y 460.597,Z 200.425,A -85,B 0,C 180,E1 -8115.998,E2 -8115.998} C_VEL
LIN {X 0,Y 460.568,Z 200.411,A -85,B 0,C 180,E1 -8118.902,E2 -8118.902} C_VEL
LIN {X 0,Y 460.513,Z 200.431,A -85,B 0,C 180,E1 -8121.486,E2 -8121.486} C_VEL
LIN {X 0,Y 460.54,Z 200.421,A -85,B 0,C 180,E1 -8124.332,E2 -8124.332} C_VEL
LIN {X 0,Y 460.577,Z 200.419,A -85,B 0,C 180,E1 -8127.243,E2 -8127.243} C_VEL
LIN {X 0,Y 460.524,Z 200.427,A -85,B 0,C 180,E1 -8130.239,E2 -8130.239} C_VEL
LIN {X 0,Y 460.527,Z 200.425,A -85,B 0,C 180,E1 -8133.325,E2 -8133.325} C_VEL
LIN {X 0,Y 460.476,Z 200.433,A -85,B 0,C 180,E1 -8136.529,E2 -8136.529} C_VEL
LIN {X 0,Y 460.555,Z 200.43,A -85,B 0,C 180,E1 -8139.86,E2 -8139.86} C_VEL
LIN {X 0,Y 460.51,Z 200.429,A -85,B 0,C 180,E1 -8142.9,E2 -8142.9} C_VEL
LIN {X 0,Y 460.507,Z 200.436,A -85,B 0,C 180,E1 -8145.831,E2 -8145.831} C_VEL
LIN {X 0,Y 460.528,Z 200.426,A -85,B 0,C 180,E1 -8148.989,E2 -8148.989} C_VEL
LIN {X 0,Y 460.517,Z 200.435,A -85,B 0,C 180,E1 -8151.266,E2 -8151.266} C_VEL
LIN {X 0,Y 460.509,Z 200.425,A -85,B 0,C 180,E1 -8154.554,E2 -8154.554} C_VEL
LIN {X 0,Y 460.53,Z 200.426,A -85,B 0,C 180,E1 -8157.716,E2 -8157.716} C_VEL
LIN {X 0,Y 460.539,Z 200.43,A -85,B 0,C 180,E1 -8160.769,E2 -8160.769} C_VEL
LIN {X 0,Y 460.562,Z 200.427,A -85,B 0,C 180,E1 -8163.735,E2 -8163.735} C_VEL
LIN {X 0,Y 460.545,Z 200.424,A -85,B 0,C 180,E1 -8166.624,E2 -8166.624} C_VEL
LIN {X 0,Y 460.55,Z 200.421,A -85,B 0,C 180,E1 -8169.453,E2 -8169.453} C_VEL
LIN {X 0,Y 460.549,Z 200.422,A -85,B 0,C 180,E1 -8172.23,E2 -8172.23} C_VEL
LIN {X 0,Y 460.564,Z 200.421,A -85,B 0,C 180,E1 -8174.965,E2 -8174.965} C_VEL
LIN {X 0,Y 460.611,Z 200.424,A -85,B 0,C 180,E1 -8178.559,E2 -8178.559} C_VEL
LIN {X 0,Y 460.576,Z 200.425,A -85,B 0,C 180,E1 -8179.23,E2 -8179.23} C_VEL
LIN {X 0,Y 459.915,Z 200.509,A -85,B 0,C 180,E1 -8179.96,E2 -8179.96} C_VEL
LIN {X 0,Y 457.072,Z 200.863,A -85,B 0,C 180,E1 -8181.146,E2 -8181.146} C_VEL
LIN {X 0,Y 454.679,Z 201.162,A -85,B 0,C 180,E1 -8182.102,E2 -8182.102} C_VEL
LIN {X 0,Y 453.669,Z 201.279,A -85,B 0,C 180,E1 -8182.841,E2 -8182.841} C_VEL
LIN {X 0,Y 453.596,Z 201.286,A -85,B 0,C 180,E1 -8183.092,E2 -8183.092} C_VEL
LIN {X 0,Y 453.655,Z 201.287,A -85,B 0,C 180,E1 -8184.499,E2 -8184.499} C_VEL
LIN {X 0,Y 455.912,Z 209.308,A -85,B 0,C 180,E1 -8185.702,E2 -8185.702} C_VEL
LIN {X 0,Y 463.163,Z 223.955,A -85,B 0,C 180,E1 -8186.478,E2 -8186.478} C_VEL
LIN {X 0,Y 467.682,Z 233.859,A -85,B 0,C 180,E1 -8186.961,E2 -8186.961} C_VEL
LIN {X 0,Y 464.687,Z 414.38,A -85,B 0,C 180,E1 -8189.911,E2 -8189.911} C_VEL
LIN {X 0,Y 464.098,Z 430.632,A -85,B 0,C 180,E1 -8190.337,E2 -8190.337} C_VEL
LIN {X 0,Y 463.284,Z 446.585,A -85,B 0,C 180,E1 -8190.923,E2 -8190.923} C_VEL
LIN {X 0,Y 462.422,Z 461.424,A -85,B 0,C 180,E1 -8191.633,E2 -8191.633} C_VEL
LIN {X 0,Y 461.337,Z 476.137,A -85,B 0,C 180,E1 -8192.51,E2 -8192.51} C_VEL
LIN {X 0,Y 460.236,Z 489.815,A -85,B 0,C 180,E1 -8193.502,E2 -8193.502} C_VEL
LIN {X 0,Y 458.969,Z 504.239,A -85,B 0,C 180,E1 -8194.75,E2 -8194.75} C_VEL
LIN {X 0,Y 457.894,Z 515.991,A -85,B 0,C 180,E1 -8195.946,E2 -8195.946} C_VEL
LIN {X 0,Y 456.658,Z 529.002,A -85,B 0,C 180,E1 -8197.516,E2 -8197.516} C_VEL
LIN {X 0,Y 455.725,Z 538.582,A -85,B 0,C 180,E1 -8198.871,E2 -8198.871} C_VEL
LIN {X 0,Y 454.876,Z 548.338,A -85,B 0,C 180,E1 -8200.459,E2 -8200.459} C_VEL
LIN {X 0,Y 454.091,Z 557.794,A -85,B 0,C 180,E1 -8202.287,E2 -8202.287} C_VEL
LIN {X 0,Y 453.542,Z 564.791,A -85,B 0,C 180,E1 -8203.897,E2 -8203.897} C_VEL
LIN {X 0,Y 452.999,Z 571.967,A -85,B 0,C 180,E1 -8205.869,E2 -8205.869} C_VEL
LIN {X 0,Y 452.794,Z 577.101,A -85,B 0,C 180,E1 -8207.617,E2 -8207.617} C_VEL
LIN {X 0,Y 452.641,Z 580.504,A -85,B 0,C 180,E1 -8209.029,E2 -8209.029} C_VEL
LIN {X 0,Y 452.401,Z 584.486,A -85,B 0,C 180,E1 -8211.237,E2 -8211.237} C_VEL
LIN {X 0,Y 452.289,Z 587.018,A -85,B 0,C 180,E1 -8213.54,E2 -8213.54} C_VEL
LIN {X 0,Y 452.266,Z 587.745,A -85,B 0,C 180,E1 -8214.807,E2 -8214.807} C_VEL
LIN {X 0,Y 452.284,Z 587.863,A -85,B 0,C 180,E1 -8216.783,E2 -8216.783} C_VEL
LIN {X 0,Y 452.313,Z 586.835,A -85,B 0,C 180,E1 -8218.794,E2 -8218.794} C_VEL
LIN {X 0,Y 452.456,Z 584.573,A -85,B 0,C 180,E1 -8220.836,E2 -8220.836} C_VEL
LIN {X 0,Y 452.612,Z 580.675,A -85,B 0,C 180,E1 -8223.019,E2 -8223.019} C_VEL
LIN {X 0,Y 452.894,Z 575.654,A -85,B 0,C 180,E1 -8225.04,E2 -8225.04} C_VEL
LIN {X 0,Y 453.162,Z 570.576,A -85,B 0,C 180,E1 -8226.683,E2 -8226.683} C_VEL
LIN {X 0,Y 453.71,Z 562.578,A -85,B 0,C 180,E1 -8228.783,E2 -8228.783} C_VEL
LIN {X 0,Y 454.423,Z 553.486,A -85,B 0,C 180,E1 -8230.728,E2 -8230.728} C_VEL
LIN {X 0,Y 455.36,Z 543.042,A -85,B 0,C 180,E1 -8232.576,E2 -8232.576} C_VEL
LIN {X 0,Y 456.381,Z 532.33,A -85,B 0,C 180,E1 -8234.172,E2 -8234.172} C_VEL
LIN {X 0,Y 457.582,Z 519.995,A -85,B 0,C 180,E1 -8235.733,E2 -8235.733} C_VEL
LIN {X 0,Y 458.86,Z 506.521,A -85,B 0,C 180,E1 -8237.172,E2 -8237.172} C_VEL
LIN {X 0,Y 460.082,Z 493.661,A -85,B 0,C 180,E1 -8238.334,E2 -8238.334} C_VEL
LIN {X 0,Y 461.34,Z 478.023,A -85,B 0,C 180,E1 -8239.51,E2 -8239.51} C_VEL
LIN {X 0,Y 462.569,Z 462.048,A -85,B 0,C 180,E1 -8240.473,E2 -8240.473} C_VEL
LIN {X 0,Y 463.481,Z 446.023,A -85,B 0,C 180,E1 -8241.242,E2 -8241.242} C_VEL
LIN {X 0,Y 464.282,Z 430.001,A -85,B 0,C 180,E1 -8241.821,E2 -8241.821} C_VEL
LIN {X 0,Y 464.891,Z 414.078,A -85,B 0,C 180,E1 -8242.229,E2 -8242.229} C_VEL
LIN {X 0,Y 467.979,Z 235.241,A -85,B 0,C 180,E1 -8245.17,E2 -8245.17} C_VEL
LIN {X 0,Y 467.567,Z 233.339,A -85,B 0,C 180,E1 -8245.233,E2 -8245.233} C_VEL
LIN {X 0,Y 457.453,Z 212.456,A -85,B 0,C 180,E1 -8246.355,E2 -8246.355} C_VEL
LIN {X 0,Y 456.121,Z 209.594,A -85,B 0,C 180,E1 -8246.54,E2 -8246.54} C_VEL
LIN {X 0,Y 453.483,Z 201.312,A -85,B 0,C 180,E1 -8247.875,E2 -8247.875} C_VEL
LIN {X 0,Y 453.484,Z 201.31,A -85,B 0,C 180,E1 -8251.287,E2 -8251.287} C_VEL
LIN {X 0,Y 453.486,Z 201.31,A -85,B 0,C 180,E1 -8254.282,E2 -8254.282} C_VEL
LIN {X 0,Y 453.471,Z 201.309,A -85,B 0,C 180,E1 -8257.204,E2 -8257.204} C_VEL
LIN {X 0,Y 453.497,Z 201.308,A -85,B 0,C 180,E1 -8260.066,E2 -8260.066} C_VEL
LIN {X 0,Y 453.492,Z 201.31,A -85,B 0,C 180,E1 -8262.875,E2 -8262.875} C_VEL
LIN {X 0,Y 453.505,Z 201.305,A -85,B 0,C 180,E1 -8265.644,E2 -8265.644} C_VEL
LIN {X 0,Y 453.552,Z 201.293,A -85,B 0,C 180,E1 -8268.379,E2 -8268.379} C_VEL
LIN {X 0,Y 453.579,Z 201.296,A -85,B 0,C 180,E1 -8271.086,E2 -8271.086} C_VEL
LIN {X 0,Y 453.658,Z 201.284,A -85,B 0,C 180,E1 -8273.774,E2 -8273.774} C_VEL
LIN {X 0,Y 453.737,Z 201.275,A -85,B 0,C 180,E1 -8277.337,E2 -8277.337} C_VEL
LIN {X 0,Y 453.816,Z 201.27,A -85,B 0,C 180,E1 -8280,E2 -8280} C_VEL
LIN {X 0,Y 453.737,Z 201.275,A -85,B 0,C 180,E1 -8282.663,E2 -8282.663} C_VEL
LIN {X 0,Y 453.67,Z 201.287,A -85,B 0,C 180,E1 -8286.225,E2 -8286.225} C_VEL
LIN {X 0,Y 453.586,Z 201.294,A -85,B 0,C 180,E1 -8288.913,E2 -8288.913} C_VEL
LIN {X 0,Y 453.557,Z 201.299,A -85,B 0,C 180,E1 -8292.529,E2 -8292.529} C_VEL
LIN {X 0,Y 453.538,Z 201.301,A -85,B 0,C 180,E1 -8296.196,E2 -8296.196} C_VEL
LIN {X 0,Y 453.514,Z 201.301,A -85,B 0,C 180,E1 -8299.041,E2 -8299.041} C_VEL
LIN {X 0,Y 453.47,Z 201.311,A -85,B 0,C 180,E1 -8301.836,E2 -8301.836} C_VEL
LIN {X 0,Y 453.508,Z 201.303,A -85,B 0,C 180,E1 -8304.735,E2 -8304.735} C_VEL
LIN {X 0,Y 453.531,Z 201.304,A -85,B 0,C 180,E1 -8307.961,E2 -8307.961} C_VEL
LIN {X 0,Y 453.461,Z 201.314,A -85,B 0,C 180,E1 -8311.526,E2 -8311.526} C_VEL
LIN {X 0,Y 453.482,Z 201.311,A -85,B 0,C 180,E1 -8314.778,E2 -8314.778} C_VEL
LIN {X 0,Y 453.459,Z 201.313,A -85,B 0,C 180,E1 -8318.312,E2 -8318.312} C_VEL
LIN {X 0,Y 453.489,Z 201.311,A -85,B 0,C 180,E1 -8320.609,E2 -8320.609} C_VEL
LIN {X 0,Y 453.451,Z 201.32,A -85,B 0,C 180,E1 -8323.245,E2 -8323.245} C_VEL
LIN {X 0,Y 453.461,Z 201.316,A -85,B 0,C 180,E1 -8325.779,E2 -8325.779} C_VEL
LIN {X 0,Y 453.474,Z 201.313,A -85,B 0,C 180,E1 -8328.21,E2 -8328.21} C_VEL
LIN {X 0,Y 453.49,Z 201.311,A -85,B 0,C 180,E1 -8330.794,E2 -8330.794} C_VEL
LIN {X 0,Y 453.45,Z 201.315,A -85,B 0,C 180,E1 -8333.918,E2 -8333.918} C_VEL
LIN {X 0,Y 453.502,Z 201.341,A -85,B 0,C 180,E1 -8335.755,E2 -8335.755} C_VEL
LIN {X 0,Y 459.216,Z 219.101,A -85,B 0,C 180,E1 -8338.346,E2 -8338.346} C_VEL
LIN {X 0,Y 462.726,Z 231.555,A -85,B 0,C 180,E1 -8340.025,E2 -8340.025} C_VEL
LIN {X 0,Y 467.628,Z 259.533,A -85,B 0,C 180,E1 -8340.875,E2 -8340.875} C_VEL
LIN {X 0,Y 465.958,Z 354.772,A -85,B 0,C 180,E1 -8342.429,E2 -8342.429} C_VEL
LIN {X 0,Y 464.631,Z 438.13,A -85,B 0,C 180,E1 -8343.808,E2 -8343.808} C_VEL
LIN {X 0,Y 463.906,Z 454.002,A -85,B 0,C 180,E1 -8344.21,E2 -8344.21} C_VEL
LIN {X 0,Y 463.089,Z 470.128,A -85,B 0,C 180,E1 -8344.794,E2 -8344.794} C_VEL
LIN {X 0,Y 462.006,Z 485.497,A -85,B 0,C 180,E1 -8345.511,E2 -8345.511} C_VEL
LIN {X 0,Y 460.905,Z 500.847,A -85,B 0,C 180,E1 -8346.426,E2 -8346.426} C_VEL
LIN {X 0,Y 459.689,Z 514.516,A -85,B 0,C 180,E1 -8347.411,E2 -8347.411} C_VEL
LIN {X 0,Y 458.361,Z 528.883,A -85,B 0,C 180,E1 -8348.645,E2 -8348.645} C_VEL
LIN {X 0,Y 457.221,Z 541.431,A -85,B 0,C 180,E1 -8349.919,E2 -8349.919} C_VEL
LIN {X 0,Y 456.174,Z 553.423,A -85,B 0,C 180,E1 -8351.357,E2 -8351.357} C_VEL
LIN {X 0,Y 455.103,Z 564.711,A -85,B 0,C 180,E1 -8352.938,E2 -8352.938} C_VEL
LIN {X 0,Y 454.259,Z 575.655,A -85,B 0,C 180,E1 -8354.752,E2 -8354.752} C_VEL
LIN {X 0,Y 453.563,Z 584.856,A -85,B 0,C 180,E1 -8356.561,E2 -8356.561} C_VEL
LIN {X 0,Y 453.139,Z 592.56,A -85,B 0,C 180,E1 -8358.368,E2 -8358.368} C_VEL
LIN {X 0,Y 452.712,Z 600.3,A -85,B 0,C 180,E1 -8360.619,E2 -8360.619} C_VEL
LIN {X 0,Y 452.568,Z 606.192,A -85,B 0,C 180,E1 -8362.864,E2 -8362.864} C_VEL
LIN {X 0,Y 452.496,Z 609.641,A -85,B 0,C 180,E1 -8364.653,E2 -8364.653} C_VEL
LIN {X 0,Y 452.428,Z 612.148,A -85,B 0,C 180,E1 -8366.438,E2 -8366.438} C_VEL
LIN {X 0,Y 452.451,Z 613.568,A -85,B 0,C 180,E1 -8368.22,E2 -8368.22} C_VEL
LIN {X 0,Y 452.43,Z 614.106,A -85,B 0,C 180,E1 -8370,E2 -8370} C_VEL
LIN {X 0,Y 452.451,Z 613.582,A -85,B 0,C 180,E1 -8371.78,E2 -8371.78} C_VEL
LIN {X 0,Y 452.428,Z 612.176,A -85,B 0,C 180,E1 -8373.563,E2 -8373.563} C_VEL
LIN {X 0,Y 452.496,Z 609.684,A -85,B 0,C 180,E1 -8375.347,E2 -8375.347} C_VEL
LIN {X 0,Y 452.569,Z 606.25,A -85,B 0,C 180,E1 -8377.137,E2 -8377.137} C_VEL
LIN {X 0,Y 452.718,Z 600.375,A -85,B 0,C 180,E1 -8379.381,E2 -8379.381} C_VEL
LIN {X 0,Y 453.143,Z 592.646,A -85,B 0,C 180,E1 -8381.632,E2 -8381.632} C_VEL
LIN {X 0,Y 453.658,Z 583.929,A -85,B 0,C 180,E1 -8383.665,E2 -8383.665} C_VEL
LIN {X 0,Y 454.415,Z 574.513,A -85,B 0,C 180,E1 -8385.473,E2 -8385.473} C_VEL
LIN {X 0,Y 455.157,Z 564.806,A -85,B 0,C 180,E1 -8387.06,E2 -8387.06} C_VEL
LIN {X 0,Y 456.156,Z 553.494,A -85,B 0,C 180,E1 -8388.645,E2 -8388.645} C_VEL
LIN {X 0,Y 457.241,Z 541.493,A -85,B 0,C 180,E1 -8390.08,E2 -8390.08} C_VEL
LIN {X 0,Y 458.485,Z 527.716,A -85,B 0,C 180,E1 -8391.468,E2 -8391.468} C_VEL
LIN {X 0,Y 459.653,Z 514.454,A -85,B 0,C 180,E1 -8392.591,E2 -8392.591} C_VEL
LIN {X 0,Y 460.981,Z 499.597,A -85,B 0,C 180,E1 -8393.642,E2 -8393.642} C_VEL
LIN {X 0,Y 462.044,Z 485.202,A -85,B 0,C 180,E1 -8394.487,E2 -8394.487} C_VEL
LIN {X 0,Y 463.137,Z 468.314,A -85,B 0,C 180,E1 -8395.264,E2 -8395.264} C_VEL
LIN {X 0,Y 463.846,Z 452.148,A -85,B 0,C 180,E1 -8395.824,E2 -8395.824} C_VEL
LIN {X 0,Y 464.593,Z 435.283,A -85,B 0,C 180,E1 -8396.215,E2 -8396.215} C_VEL
LIN {X 0,Y 467.423,Z 259.351,A -85,B 0,C 180,E1 -8399.08,E2 -8399.08} C_VEL
LIN {X 0,Y 462.619,Z 231.833,A -85,B 0,C 180,E1 -8399.909,E2 -8399.909} C_VEL
LIN {X 0,Y 459.509,Z 220.442,A -85,B 0,C 180,E1 -8401.423,E2 -8401.423} C_VEL
LIN {X 0,Y 453.514,Z 201.304,A -85,B 0,C 180,E1 -8404.144,E2 -8404.144} C_VEL
LIN {X 0,Y 453.445,Z 201.313,A -85,B 0,C 180,E1 -8407.772,E2 -8407.772} C_VEL
LIN {X 0,Y 453.491,Z 201.305,A -85,B 0,C 180,E1 -8410.609,E2 -8410.609} C_VEL
LIN {X 0,Y 453.457,Z 201.312,A -85,B 0,C 180,E1 -8414.222,E2 -8414.222} C_VEL
LIN {X 0,Y 453.445,Z 201.315,A -85,B 0,C 180,E1 -8417.003,E2 -8417.003} C_VEL
LIN {X 0,Y 453.491,Z 201.303,A -85,B 0,C 180,E1 -8419.409,E2 -8419.409} C_VEL
LIN {X 0,Y 453.449,Z 201.309,A -85,B 0,C 180,E1 -8422.81,E2 -8422.81} C_VEL
LIN {X 0,Y 453.465,Z 201.31,A -85,B 0,C 180,E1 -8426.086,E2 -8426.086} C_VEL
LIN {X 0,Y 453.473,Z 201.307,A -85,B 0,C 180,E1 -8429.24,E2 -8429.24} C_VEL
LIN {X 0,Y 453.533,Z 201.303,A -85,B 0,C 180,E1 -8432.297,E2 -8432.297} C_VEL
LIN {X 0,Y 453.497,Z 201.303,A -85,B 0,C 180,E1 -8435.265,E2 -8435.265} C_VEL
LIN {X 0,Y 453.477,Z 201.312,A -85,B 0,C 180,E1 -8438.415,E2 -8438.415} C_VEL
LIN {X 0,Y 453.519,Z 201.291,A -85,B 0,C 180,E1 -8441.009,E2 -8441.009} C_VEL
LIN {X 0,Y 453.566,Z 201.296,A -85,B 0,C 180,E1 -8443.88,E2 -8443.88} C_VEL
LIN {X 0,Y 453.561,Z 201.283,A -85,B 0,C 180,E1 -8447.471,E2 -8447.471} C_VEL
LIN {X 0,Y 453.583,Z 201.293,A -85,B 0,C 180,E1 -8451.086,E2 -8451.086} C_VEL
LIN {X 0,Y 453.662,Z 201.284,A -85,B 0,C 180,E1 -8453.775,E2 -8453.775} C_VEL
LIN {X 0,Y 453.739,Z 201.251,A -85,B 0,C 180,E1 -8457.337,E2 -8457.337} C_VEL
LIN {X 0,Y 453.819,Z 201.262,A -85,B 0,C 180,E1 -8460,E2 -8460} C_VEL
LIN {X 0,Y 453.74,Z 201.274,A -85,B 0,C 180,E1 -8462.663,E2 -8462.663} C_VEL
LIN {X 0,Y 453.673,Z 201.278,A -85,B 0,C 180,E1 -8466.225,E2 -8466.225} C_VEL
LIN {X 0,Y 453.588,Z 201.293,A -85,B 0,C 180,E1 -8468.913,E2 -8468.913} C_VEL
LIN {X 0,Y 453.561,Z 201.292,A -85,B 0,C 180,E1 -8472.529,E2 -8472.529} C_VEL
LIN {X 0,Y 453.542,Z 201.3,A -85,B 0,C 180,E1 -8476.196,E2 -8476.196} C_VEL
LIN {X 0,Y 453.517,Z 201.289,A -85,B 0,C 180,E1 -8479.041,E2 -8479.041} C_VEL
LIN {X 0,Y 453.474,Z 201.312,A -85,B 0,C 180,E1 -8481.836,E2 -8481.836} C_VEL
LIN {X 0,Y 453.511,Z 201.294,A -85,B 0,C 180,E1 -8484.734,E2 -8484.734} C_VEL
LIN {X 0,Y 453.536,Z 201.306,A -85,B 0,C 180,E1 -8487.961,E2 -8487.961} C_VEL
LIN {X 0,Y 453.481,Z 201.302,A -85,B 0,C 180,E1 -8490.759,E2 -8490.759} C_VEL
LIN {X 0,Y 453.476,Z 201.312,A -85,B 0,C 180,E1 -8493.913,E2 -8493.913} C_VEL
LIN {X 0,Y 453.468,Z 201.308,A -85,B 0,C 180,E1 -8497.188,E2 -8497.188} C_VEL
LIN {X 0,Y 453.514,Z 201.3,A -85,B 0,C 180,E1 -8499.447,E2 -8499.447} C_VEL
LIN {X 0,Y 453.46,Z 201.308,A -85,B 0,C 180,E1 -8502.995,E2 -8502.995} C_VEL
LIN {X 0,Y 453.461,Z 201.314,A -85,B 0,C 180,E1 -8505.779,E2 -8505.779} C_VEL
LIN {X 0,Y 453.477,Z 201.302,A -85,B 0,C 180,E1 -8508.209,E2 -8508.209} C_VEL
LIN {X 0,Y 453.485,Z 201.306,A -85,B 0,C 180,E1 -8510.795,E2 -8510.795} C_VEL
LIN {X 0,Y 453.453,Z 201.305,A -85,B 0,C 180,E1 -8513.917,E2 -8513.917} C_VEL
LIN {X 0,Y 453.482,Z 201.313,A -85,B 0,C 180,E1 -8517.151,E2 -8517.151} C_VEL
LIN {X 0,Y 453.474,Z 201.308,A -85,B 0,C 180,E1 -8520.268,E2 -8520.268} C_VEL
LIN {X 0,Y 453.506,Z 201.304,A -85,B 0,C 180,E1 -8523.294,E2 -8523.294} C_VEL
LIN {X 0,Y 453.502,Z 201.3,A -85,B 0,C 180,E1 -8526.239,E2 -8526.239} C_VEL
LIN {X 0,Y 453.482,Z 201.306,A -85,B 0,C 180,E1 -8529.118,E2 -8529.118} C_VEL
LIN {X 0,Y 453.503,Z 201.297,A -85,B 0,C 180,E1 -8531.944,E2 -8531.944} C_VEL
LIN {X 0,Y 453.539,Z 201.301,A -85,B 0,C 180,E1 -8534.726,E2 -8534.726} C_VEL
LIN {X 0,Y 453.56,Z 201.301,A -85,B 0,C 180,E1 -8538.379,E2 -8538.379} C_VEL
LIN {X 0,Y 453.592,Z 201.296,A -85,B 0,C 180,E1 -8541.086,E2 -8541.086} C_VEL
LIN {X 0,Y 453.596,Z 201.286,A -85,B 0,C 180,E1 -8543.092,E2 -8543.092} C_VEL
LIN {X 0,Y 453.474,Z 201.881,A -85,B 0,C 180,E1 -8543.561,E2 -8543.561} C_VEL
LIN {X 0,Y 453.092,Z 203.911,A -85,B 0,C 180,E1 -8544.103,E2 -8544.103} C_VEL
LIN {X 0,Y 452.686,Z 206.893,A -85,B 0,C 180,E1 -8544.584,E2 -8544.584} C_VEL
LIN {X 0,Y 452.481,Z 211.343,A -85,B 0,C 180,E1 -8545.085,E2 -8545.085} C_VEL
LIN {X 0,Y 452.964,Z 216.319,A -85,B 0,C 180,E1 -8545.505,E2 -8545.505} C_VEL
LIN {X 0,Y 453.943,Z 219.714,A -85,B 0,C 180,E1 -8545.736,E2 -8545.736} C_VEL
LIN {X 0,Y 454.696,Z 221.38,A -85,B 0,C 180,E1 -8545.834,E2 -8545.834} C_VEL
LIN {X 0,Y 461.412,Z 235.743,A -85,B 0,C 180,E1 -8546.566,E2 -8546.566} C_VEL
LIN {X 0,Y 458.302,Z 414.695,A -85,B 0,C 180,E1 -8549.533,E2 -8549.533} C_VEL
LIN {X 0,Y 457.665,Z 431.162,A -85,B 0,C 180,E1 -8549.972,E2 -8549.972} C_VEL
LIN {X 0,Y 456.839,Z 446.487,A -85,B 0,C 180,E1 -8550.542,E2 -8550.542} C_VEL
LIN {X 0,Y 455.997,Z 460.562,A -85,B 0,C 180,E1 -8551.214,E2 -8551.214} C_VEL
LIN {X 0,Y 454.721,Z 477.166,A -85,B 0,C 180,E1 -8552.214,E2 -8552.214} C_VEL
LIN {X 0,Y 453.419,Z 492.116,A -85,B 0,C 180,E1 -8553.332,E2 -8553.332} C_VEL
LIN {X 0,Y 452.174,Z 505.857,A -85,B 0,C 180,E1 -8554.57,E2 -8554.57} C_VEL
LIN {X 0,Y 450.79,Z 519.6,A -85,B 0,C 180,E1 -8556.04,E2 -8556.04} C_VEL
LIN {X 0,Y 449.719,Z 530.493,A -85,B 0,C 180,E1 -8557.407,E2 -8557.407} C_VEL
LIN {X 0,Y 448.667,Z 541.372,A -85,B 0,C 180,E1 -8559.012,E2 -8559.012} C_VEL
LIN {X 0,Y 447.774,Z 550.711,A -85,B 0,C 180,E1 -8560.627,E2 -8560.627} C_VEL
LIN {X 0,Y 446.952,Z 559.842,A -85,B 0,C 180,E1 -8562.486,E2 -8562.486} C_VEL
LIN {X 0,Y 446.407,Z 566.618,A -85,B 0,C 180,E1 -8564.124,E2 -8564.124} C_VEL
LIN {X 0,Y 445.931,Z 572.983,A -85,B 0,C 180,E1 -8565.977,E2 -8565.977} C_VEL
LIN {X 0,Y 445.678,Z 578.364,A -85,B 0,C 180,E1 -8567.908,E2 -8567.908} C_VEL
LIN {X 0,Y 445.5,Z 581.537,A -85,B 0,C 180,E1 -8569.346,E2 -8569.346} C_VEL
LIN {X 0,Y 445.32,Z 584.99,A -85,B 0,C 180,E1 -8571.389,E2 -8571.389} C_VEL
LIN {X 0,Y 445.183,Z 587.375,A -85,B 0,C 180,E1 -8573.705,E2 -8573.705} C_VEL
LIN {X 0,Y 445.167,Z 588.161,A -85,B 0,C 180,E1 -8575.858,E2 -8575.858} C_VEL
LIN {X 0,Y 445.222,Z 587.672,A -85,B 0,C 180,E1 -8577.874,E2 -8577.874} C_VEL
LIN {X 0,Y 445.291,Z 586.202,A -85,B 0,C 180,E1 -8579.766,E2 -8579.766} C_VEL
LIN {X 0,Y 445.397,Z 583.758,A -85,B 0,C 180,E1 -8581.562,E2 -8581.562} C_VEL
LIN {X 0,Y 445.596,Z 580.055,A -85,B 0,C 180,E1 -8583.505,E2 -8583.505} C_VEL
LIN {X 0,Y 445.872,Z 575.641,A -85,B 0,C 180,E1 -8585.268,E2 -8585.268} C_VEL
LIN {X 0,Y 446.241,Z 569.146,A -85,B 0,C 180,E1 -8587.325,E2 -8587.325} C_VEL
LIN {X 0,Y 446.851,Z 561.444,A -85,B 0,C 180,E1 -8589.295,E2 -8589.295} C_VEL
LIN {X 0,Y 447.567,Z 553.047,A -85,B 0,C 180,E1 -8591.086,E2 -8591.086} C_VEL
LIN {X 0,Y 448.59,Z 542.297,A -85,B 0,C 180,E1 -8592.997,E2 -8592.997} C_VEL
LIN {X 0,Y 449.753,Z 530.958,A -85,B 0,C 180,E1 -8594.682,E2 -8594.682} C_VEL
LIN {X 0,Y 451.07,Z 518.316,A -85,B 0,C 180,E1 -8596.265,E2 -8596.265} C_VEL
LIN {X 0,Y 452.303,Z 506.062,A -85,B 0,C 180,E1 -8597.566,E2 -8597.566} C_VEL
LIN {X 0,Y 453.547,Z 493.332,A -85,B 0,C 180,E1 -8598.723,E2 -8598.723} C_VEL
LIN {X 0,Y 454.727,Z 479.42,A -85,B 0,C 180,E1 -8599.785,E2 -8599.785} C_VEL
LIN {X 0,Y 455.891,Z 464.96,A -85,B 0,C 180,E1 -8600.693,E2 -8600.693} C_VEL
LIN {X 0,Y 456.946,Z 448.591,A -85,B 0,C 180,E1 -8601.52,E2 -8601.52} C_VEL
LIN {X 0,Y 457.807,Z 432.733,A -85,B 0,C 180,E1 -8602.132,E2 -8602.132} C_VEL
LIN {X 0,Y 458.545,Z 416.02,A -85,B 0,C 180,E1 -8602.587,E2 -8602.587} C_VEL
LIN {X 0,Y 461.767,Z 236.242,A -85,B 0,C 180,E1 -8605.6,E2 -8605.6} C_VEL
LIN {X 0,Y 452.205,Z 216.393,A -85,B 0,C 180,E1 -8606.688,E2 -8606.688} C_VEL
LIN {X 0,Y 448.85,Z 209.9,A -85,B 0,C 180,E1 -8607.103,E2 -8607.103} C_VEL
LIN {X 0,Y 446.438,Z 202.192,A -85,B 0,C 180,E1 -8608.407,E2 -8608.407} C_VEL
LIN {X 0,Y 446.442,Z 202.188,A -85,B 0,C 180,E1 -8611.83,E2 -8611.83} C_VEL
LIN {X 0,Y 446.414,Z 202.189,A -85,B 0,C 180,E1 -8614.845,E2 -8614.845} C_VEL
LIN {X 0,Y 446.441,Z 202.181,A -85,B 0,C 180,E1 -8618.245,E2 -8618.245} C_VEL
LIN {X 0,Y 446.445,Z 202.185,A -85,B 0,C 180,E1 -8621.649,E2 -8621.649} C_VEL
LIN {X 0,Y 446.501,Z 202.173,A -85,B 0,C 180,E1 -8624.48,E2 -8624.48} C_VEL
LIN {X 0,Y 446.51,Z 202.169,A -85,B 0,C 180,E1 -8628.193,E2 -8628.193} C_VEL
LIN {X 0,Y 446.526,Z 202.175,A -85,B 0,C 180,E1 -8630.944,E2 -8630.944} C_VEL
LIN {X 0,Y 446.627,Z 202.159,A -85,B 0,C 180,E1 -8633.676,E2 -8633.676} C_VEL
LIN {X 0,Y 446.684,Z 202.154,A -85,B 0,C 180,E1 -8637.295,E2 -8637.295} C_VEL
LIN {X 0,Y 446.786,Z 202.146,A -85,B 0,C 180,E1 -8640,E2 -8640} C_VEL
LIN {X 0,Y 446.684,Z 202.153,A -85,B 0,C 180,E1 -8642.705,E2 -8642.705} C_VEL
LIN {X 0,Y 446.639,Z 202.164,A -85,B 0,C 180,E1 -8646.324,E2 -8646.324} C_VEL
LIN {X 0,Y 446.531,Z 202.172,A -85,B 0,C 180,E1 -8649.055,E2 -8649.055} C_VEL
LIN {X 0,Y 446.515,Z 202.175,A -85,B 0,C 180,E1 -8652.73,E2 -8652.73} C_VEL
LIN {X 0,Y 446.49,Z 202.179,A -85,B 0,C 180,E1 -8656.228,E2 -8656.228} C_VEL
LIN {X 0,Y 446.463,Z 202.181,A -85,B 0,C 180,E1 -8659.303,E2 -8659.303} C_VEL
LIN {X 0,Y 446.413,Z 202.191,A -85,B 0,C 180,E1 -8662.2,E2 -8662.2} C_VEL
LIN {X 0,Y 446.452,Z 202.184,A -85,B 0,C 180,E1 -8665.152,E2 -8665.152} C_VEL
LIN {X 0,Y 446.478,Z 202.181,A -85,B 0,C 180,E1 -8668.179,E2 -8668.179} C_VEL
LIN {X 0,Y 446.414,Z 202.192,A -85,B 0,C 180,E1 -8671.775,E2 -8671.775} C_VEL
LIN {X 0,Y 446.423,Z 202.189,A -85,B 0,C 180,E1 -8674.523,E2 -8674.523} C_VEL
LIN {X 0,Y 446.41,Z 202.192,A -85,B 0,C 180,E1 -8678.08,E2 -8678.08} C_VEL
LIN {X 0,Y 446.422,Z 202.194,A -85,B 0,C 180,E1 -8680.918,E2 -8680.918} C_VEL
LIN {X 0,Y 446.397,Z 202.195,A -85,B 0,C 180,E1 -8683.846,E2 -8683.846} C_VEL
LIN {X 0,Y 446.395,Z 202.196,A -85,B 0,C 180,E1 -8686.404,E2 -8686.404} C_VEL
LIN {X 0,Y 446.422,Z 202.192,A -85,B 0,C 180,E1 -8689.083,E2 -8689.083} C_VEL
LIN {X 0,Y 446.405,Z 202.191,A -85,B 0,C 180,E1 -8692.122,E2 -8692.122} C_VEL
LIN {X 0,Y 446.464,Z 202.242,A -85,B 0,C 180,E1 -8695.256,E2 -8695.256} C_VEL
LIN {X 0,Y 452.302,Z 220.277,A -85,B 0,C 180,E1 -8697.956,E2 -8697.956} C_VEL
LIN {X 0,Y 455.48,Z 231.21,A -85,B 0,C 180,E1 -8699.48,E2 -8699.48} C_VEL
LIN {X 0,Y 457.02,Z 234.929,A -85,B 0,C 180,E1 -8699.665,E2 -8699.665} C_VEL
LIN {X 0,Y 461.439,Z 260.544,A -85,B 0,C 180,E1 -8700.455,E2 -8700.455} C_VEL
LIN {X 0,Y 459.239,Z 382.082,A -85,B 0,C 180,E1 -8702.471,E2 -8702.471} C_VEL
LIN {X 0,Y 458.283,Z 438.41,A -85,B 0,C 180,E1 -8703.423,E2 -8703.423} C_VEL
LIN {X 0,Y 457.516,Z 453.901,A -85,B 0,C 180,E1 -8703.823,E2 -8703.823} C_VEL
LIN {X 0,Y 456.665,Z 469.991,A -85,B 0,C 180,E1 -8704.414,E2 -8704.414} C_VEL
LIN {X 0,Y 455.542,Z 485.339,A -85,B 0,C 180,E1 -8705.14,E2 -8705.14} C_VEL
LIN {X 0,Y 454.276,Z 501.638,A -85,B 0,C 180,E1 -8706.127,E2 -8706.127} C_VEL
LIN {X 0,Y 452.936,Z 515.774,A -85,B 0,C 180,E1 -8707.176,E2 -8707.176} C_VEL
LIN {X 0,Y 451.571,Z 529.873,A -85,B 0,C 180,E1 -8708.428,E2 -8708.428} C_VEL
LIN {X 0,Y 450.303,Z 542.754,A -85,B 0,C 180,E1 -8709.782,E2 -8709.782} C_VEL
LIN {X 0,Y 449.18,Z 554.975,A -85,B 0,C 180,E1 -8711.292,E2 -8711.292} C_VEL
LIN {X 0,Y 448.019,Z 566.656,A -85,B 0,C 180,E1 -8712.997,E2 -8712.997} C_VEL
LIN {X 0,Y 447.202,Z 576.69,A -85,B 0,C 180,E1 -8714.738,E2 -8714.738} C_VEL
LIN {X 0,Y 446.486,Z 585.664,A -85,B 0,C 180,E1 -8716.575,E2 -8716.575} C_VEL
LIN {X 0,Y 446.12,Z 592.351,A -85,B 0,C 180,E1 -8718.183,E2 -8718.183} C_VEL
LIN {X 0,Y 445.629,Z 600.09,A -85,B 0,C 180,E1 -8720.469,E2 -8720.469} C_VEL
LIN {X 0,Y 445.485,Z 605.984,A -85,B 0,C 180,E1 -8722.75,E2 -8722.75} C_VEL
LIN {X 0,Y 445.398,Z 609.434,A -85,B 0,C 180,E1 -8724.568,E2 -8724.568} C_VEL
LIN {X 0,Y 445.327,Z 611.942,A -85,B 0,C 180,E1 -8726.381,E2 -8726.381} C_VEL
LIN {X 0,Y 445.369,Z 613.363,A -85,B 0,C 180,E1 -8728.192,E2 -8728.192} C_VEL
LIN {X 0,Y 445.338,Z 613.901,A -85,B 0,C 180,E1 -8730,E2 -8730} C_VEL
LIN {X 0,Y 445.369,Z 613.377,A -85,B 0,C 180,E1 -8731.809,E2 -8731.809} C_VEL
LIN {X 0,Y 445.327,Z 611.969,A -85,B 0,C 180,E1 -8733.62,E2 -8733.62} C_VEL
LIN {X 0,Y 445.399,Z 609.475,A -85,B 0,C 180,E1 -8735.433,E2 -8735.433} C_VEL
LIN {X 0,Y 445.486,Z 606.038,A -85,B 0,C 180,E1 -8737.251,E2 -8737.251} C_VEL
LIN {X 0,Y 445.635,Z 600.157,A -85,B 0,C 180,E1 -8739.532,E2 -8739.532} C_VEL
LIN {X 0,Y 446.117,Z 592.42,A -85,B 0,C 180,E1 -8741.818,E2 -8741.818} C_VEL
LIN {X 0,Y 446.643,Z 583.694,A -85,B 0,C 180,E1 -8743.884,E2 -8743.884} C_VEL
LIN {X 0,Y 447.474,Z 574.272,A -85,B 0,C 180,E1 -8745.72,E2 -8745.72} C_VEL
LIN {X 0,Y 448.261,Z 564.556,A -85,B 0,C 180,E1 -8747.331,E2 -8747.331} C_VEL
LIN {X 0,Y 449.332,Z 553.229,A -85,B 0,C 180,E1 -8748.938,E2 -8748.938} C_VEL
LIN {X 0,Y 450.428,Z 541.622,A -85,B 0,C 180,E1 -8750.348,E2 -8750.348} C_VEL
LIN {X 0,Y 451.676,Z 528.598,A -85,B 0,C 180,E1 -8751.688,E2 -8751.688} C_VEL
LIN {X 0,Y 453.02,Z 514.131,A -85,B 0,C 180,E1 -8752.941,E2 -8752.941} C_VEL
LIN {X 0,Y 454.374,Z 499.332,A -85,B 0,C 180,E1 -8754.001,E2 -8754.001} C_VEL
LIN {X 0,Y 455.593,Z 483.695,A -85,B 0,C 180,E1 -8754.918,E2 -8754.918} C_VEL
LIN {X 0,Y 456.669,Z 467.884,A -85,B 0,C 180,E1 -8755.648,E2 -8755.648} C_VEL
LIN {X 0,Y 457.469,Z 451.618,A -85,B 0,C 180,E1 -8756.211,E2 -8756.211} C_VEL
LIN {X 0,Y 458.209,Z 434.936,A -85,B 0,C 180,E1 -8756.6,E2 -8756.6} C_VEL
LIN {X 0,Y 461.181,Z 260.506,A -85,B 0,C 180,E1 -8759.48,E2 -8759.48} C_VEL
LIN {X 0,Y 456.409,Z 233.855,A -85,B 0,C 180,E1 -8760.29,E2 -8760.29} C_VEL
LIN {X 0,Y 455.493,Z 231.57,A -85,B 0,C 180,E1 -8760.421,E2 -8760.421} C_VEL
LIN {X 0,Y 450.113,Z 213.703,A -85,B 0,C 180,E1 -8762.907,E2 -8762.907} C_VEL
LIN {X 0,Y 446.468,Z 202.187,A -85,B 0,C 180,E1 -8764.618,E2 -8764.618} C_VEL
LIN {X 0,Y 446.41,Z 202.191,A -85,B 0,C 180,E1 -8768.079,E2 -8768.079} C_VEL
LIN {X 0,Y 446.42,Z 202.189,A -85,B 0,C 180,E1 -8770.917,E2 -8770.917} C_VEL
LIN {X 0,Y 446.396,Z 202.192,A -85,B 0,C 180,E1 -8773.846,E2 -8773.846} C_VEL
LIN {X 0,Y 446.394,Z 202.186,A -85,B 0,C 180,E1 -8776.404,E2 -8776.404} C_VEL
LIN {X 0,Y 446.432,Z 202.182,A -85,B 0,C 180,E1 -8779.801,E2 -8779.801} C_VEL
LIN {X 0,Y 446.399,Z 202.183,A -85,B 0,C 180,E1 -8783.255,E2 -8783.255} C_VEL
LIN {X 0,Y 446.446,Z 202.188,A -85,B 0,C 180,E1 -8786.566,E2 -8786.566} C_VEL
LIN {X 0,Y 446.427,Z 202.183,A -85,B 0,C 180,E1 -8789.979,E2 -8789.979} C_VEL
LIN {X 0,Y 446.468,Z 202.175,A -85,B 0,C 180,E1 -8792.839,E2 -8792.839} C_VEL
LIN {X 0,Y 446.459,Z 202.179,A -85,B 0,C 180,E1 -8795.924,E2 -8795.924} C_VEL
LIN {X 0,Y 446.45,Z 202.18,A -85,B 0,C 180,E1 -8798.773,E2 -8798.773} C_VEL
LIN {X 0,Y 446.447,Z 202.172,A -85,B 0,C 180,E1 -8801.649,E2 -8801.649} C_VEL
LIN {X 0,Y 446.504,Z 202.182,A -85,B 0,C 180,E1 -8804.48,E2 -8804.48} C_VEL
LIN {X 0,Y 446.514,Z 202.158,A -85,B 0,C 180,E1 -8808.193,E2 -8808.193} C_VEL
LIN {X 0,Y 446.53,Z 202.173,A -85,B 0,C 180,E1 -8810.945,E2 -8810.945} C_VEL
LIN {X 0,Y 446.631,Z 202.16,A -85,B 0,C 180,E1 -8813.676,E2 -8813.676} C_VEL
LIN {X 0,Y 446.686,Z 202.129,A -85,B 0,C 180,E1 -8817.295,E2 -8817.295} C_VEL
LIN {X 0,Y 446.789,Z 202.137,A -85,B 0,C 180,E1 -8820,E2 -8820} C_VEL
LIN {X 0,Y 446.687,Z 202.152,A -85,B 0,C 180,E1 -8822.705,E2 -8822.705} C_VEL
LIN {X 0,Y 446.643,Z 202.155,A -85,B 0,C 180,E1 -8826.324,E2 -8826.324} C_VEL
LIN {X 0,Y 446.533,Z 202.171,A -85,B 0,C 180,E1 -8829.055,E2 -8829.055} C_VEL
LIN {X 0,Y 446.519,Z 202.167,A -85,B 0,C 180,E1 -8832.73,E2 -8832.73} C_VEL
LIN {X 0,Y 446.493,Z 202.178,A -85,B 0,C 180,E1 -8836.228,E2 -8836.228} C_VEL
LIN {X 0,Y 446.467,Z 202.168,A -85,B 0,C 180,E1 -8839.303,E2 -8839.303} C_VEL
LIN {X 0,Y 446.416,Z 202.19,A -85,B 0,C 180,E1 -8842.2,E2 -8842.2} C_VEL
LIN {X 0,Y 446.455,Z 202.173,A -85,B 0,C 180,E1 -8845.152,E2 -8845.152} C_VEL
LIN {X 0,Y 446.482,Z 202.182,A -85,B 0,C 180,E1 -8848.179,E2 -8848.179} C_VEL
LIN {X 0,Y 446.417,Z 202.184,A -85,B 0,C 180,E1 -8851.3,E2 -8851.3} C_VEL
LIN {X 0,Y 446.428,Z 202.185,A -85,B 0,C 180,E1 -8854.523,E2 -8854.523} C_VEL
LIN {X 0,Y 446.428,Z 202.178,A -85,B 0,C 180,E1 -8858.082,E2 -8858.082} C_VEL
LIN {X 0,Y 446.425,Z 202.187,A -85,B 0,C 180,E1 -8860.918,E2 -8860.918} C_VEL
LIN {X 0,Y 446.397,Z 202.185,A -85,B 0,C 180,E1 -8863.846,E2 -8863.846} C_VEL
LIN {X 0,Y 446.396,Z 202.19,A -85,B 0,C 180,E1 -8866.404,E2 -8866.404} C_VEL
LIN {X 0,Y 446.425,Z 202.182,A -85,B 0,C 180,E1 -8869.083,E2 -8869.083} C_VEL
LIN {X 0,Y 446.406,Z 202.188,A -85,B 0,C 180,E1 -8872.121,E2 -8872.121} C_VEL
LIN {X 0,Y 446.428,Z 202.189,A -85,B 0,C 180,E1 -8875.477,E2 -8875.477} C_VEL
LIN {X 0,Y 446.415,Z 202.182,A -85,B 0,C 180,E1 -8878.7,E2 -8878.7} C_VEL
LIN {X 0,Y 446.484,Z 202.177,A -85,B 0,C 180,E1 -8881.821,E2 -8881.821} C_VEL
LIN {X 0,Y 446.457,Z 202.186,A -85,B 0,C 180,E1 -8884.848,E2 -8884.848} C_VEL
LIN {X 0,Y 446.447,Z 202.185,A -85,B 0,C 180,E1 -8888.245,E2 -8888.245} C_VEL
LIN {X 0,Y 446.451,Z 202.171,A -85,B 0,C 180,E1 -8891.649,E2 -8891.649} C_VEL
LIN {X 0,Y 446.507,Z 202.181,A -85,B 0,C 180,E1 -8894.48,E2 -8894.48} C_VEL
LIN {X 0,Y 446.517,Z 202.177,A -85,B 0,C 180,E1 -8898.193,E2 -8898.193} C_VEL
LIN {X 0,Y 446.538,Z 202.175,A -85,B 0,C 180,E1 -8900.944,E2 -8900.944} C_VEL
LIN {X 0,Y 446.61,Z 202.155,A -85,B 0,C 180,E1 -8903.902,E2 -8903.902} C_VEL
LIN {X 0,Y 446.647,Z 202.315,A -85,B 0,C 180,E1 -8904.073,E2 -8904.073} C_VEL
LIN {X 0,Y 448.764,Z 209.695,A -85,B 0,C 180,E1 -8905.183,E2 -8905.183} C_VEL
LIN {X 0,Y 454.696,Z 221.38,A -85,B 0,C 180,E1 -8905.834,E2 -8905.834} C_VEL
LIN {X 0,Y 456.005,Z 224.857,A -85,B 0,C 180,E1 -8905.991,E2 -8905.991} C_VEL
LIN {X 0,Y 456.795,Z 230.584,A -85,B 0,C 180,E1 -8906.151,E2 -8906.151} C_VEL
LIN {X 0,Y 456.611,Z 236.519,A -85,B 0,C 180,E1 -8906.245,E2 -8906.245} C_VEL
LIN {X 0,Y 454.958,Z 252.973,A -85,B 0,C 180,E1 -8906.427,E2 -8906.427} C_VEL
LIN {X 0,Y 451.924,Z 414.604,A -85,B 0,C 180,E1 -8909.137,E2 -8909.137} C_VEL
LIN {X 0,Y 451.269,Z 431.167,A -85,B 0,C 180,E1 -8909.581,E2 -8909.581} C_VEL
LIN {X 0,Y 450.369,Z 447.147,A -85,B 0,C 180,E1 -8910.185,E2 -8910.185} C_VEL
LIN {X 0,Y 449.439,Z 461.669,A -85,B 0,C 180,E1 -8910.896,E2 -8910.896} C_VEL
LIN {X 0,Y 448.275,Z 476.399,A -85,B 0,C 180,E1 -8911.797,E2 -8911.797} C_VEL
LIN {X 0,Y 447.024,Z 490.149,A -85,B 0,C 180,E1 -8912.816,E2 -8912.816} C_VEL
LIN {X 0,Y 445.692,Z 504.275,A -85,B 0,C 180,E1 -8914.069,E2 -8914.069} C_VEL
LIN {X 0,Y 444.32,Z 517.367,A -85,B 0,C 180,E1 -8915.445,E2 -8915.445} C_VEL
LIN {X 0,Y 442.978,Z 530.276,A -85,B 0,C 180,E1 -8917.062,E2 -8917.062} C_VEL
LIN {X 0,Y 441.83,Z 541.207,A -85,B 0,C 180,E1 -8918.691,E2 -8918.691} C_VEL
LIN {X 0,Y 440.882,Z 550.607,A -85,B 0,C 180,E1 -8920.331,E2 -8920.331} C_VEL
LIN {X 0,Y 440.128,Z 558.763,A -85,B 0,C 180,E1 -8921.98,E2 -8921.98} C_VEL
LIN {X 0,Y 439.438,Z 566.591,A -85,B 0,C 180,E1 -8923.88,E2 -8923.88} C_VEL
LIN {X 0,Y 438.889,Z 573.112,A -85,B 0,C 180,E1 -8925.796,E2 -8925.796} C_VEL
LIN {X 0,Y 438.617,Z 578.433,A -85,B 0,C 180,E1 -8927.724,E2 -8927.724} C_VEL
LIN {X 0,Y 438.364,Z 582.57,A -85,B 0,C 180,E1 -8929.674,E2 -8929.674} C_VEL
LIN {X 0,Y 438.2,Z 585.591,A -85,B 0,C 180,E1 -8931.646,E2 -8931.646} C_VEL
LIN {X 0,Y 438.093,Z 587.687,A -85,B 0,C 180,E1 -8933.879,E2 -8933.879} C_VEL
LIN {X 0,Y 438.087,Z 588.394,A -85,B 0,C 180,E1 -8936.055,E2 -8936.055} C_VEL
LIN {X 0,Y 438.124,Z 587.788,A -85,B 0,C 180,E1 -8938.084,E2 -8938.084} C_VEL
LIN {X 0,Y 438.222,Z 586.203,A -85,B 0,C 180,E1 -8940,E2 -8940} C_VEL
LIN {X 0,Y 438.353,Z 583.518,A -85,B 0,C 180,E1 -8941.943,E2 -8941.943} C_VEL
LIN {X 0,Y 438.615,Z 579.164,A -85,B 0,C 180,E1 -8944.111,E2 -8944.111} C_VEL
LIN {X 0,Y 438.904,Z 574.915,A -85,B 0,C 180,E1 -8945.763,E2 -8945.763} C_VEL
LIN {X 0,Y 439.378,Z 567.932,A -85,B 0,C 180,E1 -8947.925,E2 -8947.925} C_VEL
LIN {X 0,Y 440.041,Z 559.783,A -85,B 0,C 180,E1 -8949.949,E2 -8949.949} C_VEL
LIN {X 0,Y 440.823,Z 551.358,A -85,B 0,C 180,E1 -8951.694,E2 -8951.694} C_VEL
LIN {X 0,Y 441.902,Z 541.316,A -85,B 0,C 180,E1 -8953.459,E2 -8953.459} C_VEL
LIN {X 0,Y 443.07,Z 530.632,A -85,B 0,C 180,E1 -8955.058,E2 -8955.058} C_VEL
LIN {X 0,Y 444.229,Z 519.848,A -85,B 0,C 180,E1 -8956.43,E2 -8956.43} C_VEL
LIN {X 0,Y 445.605,Z 506.958,A -85,B 0,C 180,E1 -8957.839,E2 -8957.839} C_VEL
LIN {X 0,Y 446.912,Z 494.382,A -85,B 0,C 180,E1 -8959.009,E2 -8959.009} C_VEL
LIN {X 0,Y 448.279,Z 479.125,A -85,B 0,C 180,E1 -8960.192,E2 -8960.192} C_VEL
LIN {X 0,Y 449.526,Z 464.186,A -85,B 0,C 180,E1 -8961.131,E2 -8961.131} C_VEL
LIN {X 0,Y 450.531,Z 449.409,A -85,B 0,C 180,E1 -8961.885,E2 -8961.885} C_VEL
LIN {X 0,Y 451.472,Z 433.185,A -85,B 0,C 180,E1 -8962.524,E2 -8962.524} C_VEL
LIN {X 0,Y 452.194,Z 416.813,A -85,B 0,C 180,E1 -8962.982,E2 -8962.982} C_VEL
LIN {X 0,Y 453.478,Z 347.496,A -85,B 0,C 180,E1 -8964.174,E2 -8964.174} C_VEL
LIN {X 0,Y 455.631,Z 238.432,A -85,B 0,C 180,E1 -8966.014,E2 -8966.014} C_VEL
LIN {X 0,Y 445.885,Z 218.189,A -85,B 0,C 180,E1 -8967.159,E2 -8967.159} C_VEL
LIN {X 0,Y 441.719,Z 210.292,A -85,B 0,C 180,E1 -8967.667,E2 -8967.667} C_VEL
LIN {X 0,Y 439.354,Z 203.071,A -85,B 0,C 180,E1 -8968.911,E2 -8968.911} C_VEL
LIN {X 0,Y 439.376,Z 203.069,A -85,B 0,C 180,E1 -8972.363,E2 -8972.363} C_VEL
LIN {X 0,Y 439.368,Z 203.067,A -85,B 0,C 180,E1 -8975.747,E2 -8975.747} C_VEL
LIN {X 0,Y 439.408,Z 203.058,A -85,B 0,C 180,E1 -8978.416,E2 -8978.416} C_VEL
LIN {X 0,Y 439.417,Z 203.059,A -85,B 0,C 180,E1 -8981.345,E2 -8981.345} C_VEL
LIN {X 0,Y 439.455,Z 203.051,A -85,B 0,C 180,E1 -8984.224,E2 -8984.224} C_VEL
LIN {X 0,Y 439.476,Z 203.045,A -85,B 0,C 180,E1 -8988.001,E2 -8988.001} C_VEL
LIN {X 0,Y 439.489,Z 203.052,A -85,B 0,C 180,E1 -8990.798,E2 -8990.798} C_VEL
LIN {X 0,Y 439.597,Z 203.035,A -85,B 0,C 180,E1 -8993.574,E2 -8993.574} C_VEL
LIN {X 0,Y 439.633,Z 203.033,A -85,B 0,C 180,E1 -8997.251,E2 -8997.251} C_VEL
LIN {X 0,Y 439.756,Z 203.021,A -85,B 0,C 180,E1 -9000,E2 -9000} C_VEL
LIN {X 0,Y 439.634,Z 203.031,A -85,B 0,C 180,E1 -9002.749,E2 -9002.749} C_VEL
LIN {X 0,Y 439.611,Z 203.04,A -85,B 0,C 180,E1 -9006.425,E2 -9006.425} C_VEL
LIN {X 0,Y 439.493,Z 203.049,A -85,B 0,C 180,E1 -9009.202,E2 -9009.202} C_VEL
LIN {X 0,Y 439.459,Z 203.054,A -85,B 0,C 180,E1 -9012.938,E2 -9012.938} C_VEL
LIN {X 0,Y 439.441,Z 203.056,A -85,B 0,C 180,E1 -9016.349,E2 -9016.349} C_VEL
LIN {X 0,Y 439.396,Z 203.063,A -85,B 0,C 180,E1 -9019.626,E2 -9019.626} C_VEL
LIN {X 0,Y 439.359,Z 203.067,A -85,B 0,C 180,E1 -9022.576,E2 -9022.576} C_VEL
LIN {X 0,Y 439.4,Z 203.067,A -85,B 0,C 180,E1 -9025.585,E2 -9025.585} C_VEL
LIN {X 0,Y 439.412,Z 203.06,A -85,B 0,C 180,E1 -9028.674,E2 -9028.674} C_VEL
LIN {X 0,Y 439.365,Z 203.07,A -85,B 0,C 180,E1 -9032.031,E2 -9032.031} C_VEL
LIN {X 0,Y 439.389,Z 203.07,A -85,B 0,C 180,E1 -9035.341,E2 -9035.341} C_VEL
LIN {X 0,Y 439.378,Z 203.068,A -85,B 0,C 180,E1 -9038.595,E2 -9038.595} C_VEL
LIN {X 0,Y 439.383,Z 203.073,A -85,B 0,C 180,E1 -9041.257,E2 -9041.257} C_VEL
LIN {X 0,Y 439.396,Z 203.07,A -85,B 0,C 180,E1 -9044.73,E2 -9044.73} C_VEL
LIN {X 0,Y 439.391,Z 203.068,A -85,B 0,C 180,E1 -9047.796,E2 -9047.796} C_VEL
LIN {X 0,Y 439.421,Z 203.062,A -85,B 0,C 180,E1 -9050.228,E2 -9050.228} C_VEL
LIN {X 0,Y 439.369,Z 203.07,A -85,B 0,C 180,E1 -9053.713,E2 -9053.713} C_VEL
LIN {X 0,Y 439.403,Z 203.259,A -85,B 0,C 180,E1 -9054.744,E2 -9054.744} C_VEL
LIN {X 0,Y 444.204,Z 217.674,A -85,B 0,C 180,E1 -9056.986,E2 -9056.986} C_VEL
LIN {X 0,Y 448.258,Z 231.087,A -85,B 0,C 180,E1 -9058.917,E2 -9058.917} C_VEL
LIN {X 0,Y 451.283,Z 238.038,A -85,B 0,C 180,E1 -9059.285,E2 -9059.285} C_VEL
LIN {X 0,Y 455.33,Z 261.829,A -85,B 0,C 180,E1 -9060.033,E2 -9060.033} C_VEL
LIN {X 0,Y 451.952,Z 438.711,A -85,B 0,C 180,E1 -9063.026,E2 -9063.026} C_VEL
LIN {X 0,Y 451.115,Z 454.726,A -85,B 0,C 180,E1 -9063.454,E2 -9063.454} C_VEL
LIN {X 0,Y 450.15,Z 471.153,A -85,B 0,C 180,E1 -9064.078,E2 -9064.078} C_VEL
LIN {X 0,Y 448.894,Z 487.172,A -85,B 0,C 180,E1 -9064.87,E2 -9064.87} C_VEL
LIN {X 0,Y 447.693,Z 501.944,A -85,B 0,C 180,E1 -9065.789,E2 -9065.789} C_VEL
LIN {X 0,Y 446.193,Z 517.034,A -85,B 0,C 180,E1 -9066.934,E2 -9066.934} C_VEL
LIN {X 0,Y 444.778,Z 530.873,A -85,B 0,C 180,E1 -9068.203,E2 -9068.203} C_VEL
LIN {X 0,Y 443.434,Z 543.701,A -85,B 0,C 180,E1 -9069.594,E2 -9069.594} C_VEL
LIN {X 0,Y 442.362,Z 554.781,A -85,B 0,C 180,E1 -9070.993,E2 -9070.993} C_VEL
LIN {X 0,Y 441.064,Z 567.042,A -85,B 0,C 180,E1 -9072.817,E2 -9072.817} C_VEL
LIN {X 0,Y 440.251,Z 576.485,A -85,B 0,C 180,E1 -9074.491,E2 -9074.491} C_VEL
LIN {X 0,Y 439.486,Z 585.459,A -85,B 0,C 180,E1 -9076.357,E2 -9076.357} C_VEL
LIN {X 0,Y 439.085,Z 592.144,A -85,B 0,C 180,E1 -9077.991,E2 -9077.991} C_VEL
LIN {X 0,Y 438.562,Z 599.883,A -85,B 0,C 180,E1 -9080.314,E2 -9080.314} C_VEL
LIN {X 0,Y 438.388,Z 605.778,A -85,B 0,C 180,E1 -9082.632,E2 -9082.632} C_VEL
LIN {X 0,Y 438.307,Z 609.229,A -85,B 0,C 180,E1 -9084.48,E2 -9084.48} C_VEL
LIN {X 0,Y 438.23,Z 611.737,A -85,B 0,C 180,E1 -9086.322,E2 -9086.322} C_VEL
LIN {X 0,Y 438.289,Z 613.159,A -85,B 0,C 180,E1 -9088.162,E2 -9088.162} C_VEL
LIN {X 0,Y 438.249,Z 613.696,A -85,B 0,C 180,E1 -9090,E2 -9090} C_VEL
LIN {X 0,Y 438.289,Z 613.171,A -85,B 0,C 180,E1 -9091.838,E2 -9091.838} C_VEL
LIN {X 0,Y 438.23,Z 611.76,A -85,B 0,C 180,E1 -9093.678,E2 -9093.678} C_VEL
LIN {X 0,Y 438.307,Z 609.264,A -85,B 0,C 180,E1 -9095.521,E2 -9095.521} C_VEL
LIN {X 0,Y 438.388,Z 605.821,A -85,B 0,C 180,E1 -9097.369,E2 -9097.369} C_VEL
LIN {X 0,Y 438.567,Z 599.935,A -85,B 0,C 180,E1 -9099.687,E2 -9099.687} C_VEL
LIN {X 0,Y 438.941,Z 593.863,A -85,B 0,C 180,E1 -9101.545,E2 -9101.545} C_VEL
LIN {X 0,Y 439.414,Z 586.525,A -85,B 0,C 180,E1 -9103.41,E2 -9103.41} C_VEL
LIN {X 0,Y 440.122,Z 577.756,A -85,B 0,C 180,E1 -9105.277,E2 -9105.277} C_VEL
LIN {X 0,Y 441.002,Z 567.99,A -85,B 0,C 180,E1 -9107.024,E2 -9107.024} C_VEL
LIN {X 0,Y 441.957,Z 558.026,A -85,B 0,C 180,E1 -9108.544,E2 -9108.544} C_VEL
LIN {X 0,Y 443.246,Z 545.558,A -85,B 0,C 180,E1 -9110.173,E2 -9110.173} C_VEL
LIN {X 0,Y 444.513,Z 533.025,A -85,B 0,C 180,E1 -9111.567,E2 -9111.567} C_VEL
LIN {X 0,Y 445.881,Z 519.41,A -85,B 0,C 180,E1 -9112.839,E2 -9112.839} C_VEL
LIN {X 0,Y 447.296,Z 504.633,A -85,B 0,C 180,E1 -9113.988,E2 -9113.988} C_VEL
LIN {X 0,Y 448.592,Z 489.986,A -85,B 0,C 180,E1 -9114.927,E2 -9114.927} C_VEL
LIN {X 0,Y 449.71,Z 475.216,A -85,B 0,C 180,E1 -9115.701,E2 -9115.701} C_VEL
LIN {X 0,Y 450.735,Z 458.285,A -85,B 0,C 180,E1 -9116.384,E2 -9116.384} C_VEL
LIN {X 0,Y 451.548,Z 441.612,A -85,B 0,C 180,E1 -9116.854,E2 -9116.854} C_VEL
LIN {X 0,Y 452.186,Z 418.47,A -85,B 0,C 180,E1 -9117.27,E2 -9117.27} C_VEL
LIN {X 0,Y 454.926,Z 261.435,A -85,B 0,C 180,E1 -9119.895,E2 -9119.895} C_VEL
LIN {X 0,Y 450.572,Z 236.7,A -85,B 0,C 180,E1 -9120.657,E2 -9120.657} C_VEL
LIN {X 0,Y 448.223,Z 231.544,A -85,B 0,C 180,E1 -9120.932,E2 -9120.932} C_VEL
LIN {X 0,Y 443.309,Z 215.227,A -85,B 0,C 180,E1 -9123.252,E2 -9123.252} C_VEL
LIN {X 0,Y 439.389,Z 203.064,A -85,B 0,C 180,E1 -9125.111,E2 -9125.111} C_VEL
LIN {X 0,Y 439.373,Z 203.069,A -85,B 0,C 180,E1 -9128.596,E2 -9128.596} C_VEL
LIN {X 0,Y 439.379,Z 203.071,A -85,B 0,C 180,E1 -9131.256,E2 -9131.256} C_VEL
LIN {X 0,Y 439.396,Z 203.066,A -85,B 0,C 180,E1 -9134.73,E2 -9134.73} C_VEL
LIN {X 0,Y 439.381,Z 203.065,A -85,B 0,C 180,E1 -9137.794,E2 -9137.794} C_VEL
LIN {X 0,Y 439.386,Z 203.06,A -85,B 0,C 180,E1 -9140.223,E2 -9140.223} C_VEL
LIN {X 0,Y 439.37,Z 203.057,A -85,B 0,C 180,E1 -9143.713,E2 -9143.713} C_VEL
LIN {X 0,Y 439.368,Z 203.062,A -85,B 0,C 180,E1 -9147.054,E2 -9147.054} C_VEL
LIN {X 0,Y 439.378,Z 203.063,A -85,B 0,C 180,E1 -9150.274,E2 -9150.274} C_VEL
LIN {X 0,Y 439.425,Z 203.047,A -85,B 0,C 180,E1 -9153.396,E2 -9153.396} C_VEL
LIN {X 0,Y 439.381,Z 203.065,A -85,B 0,C 180,E1 -9156.429,E2 -9156.429} C_VEL
LIN {X 0,Y 439.384,Z 203.055,A -85,B 0,C 180,E1 -9159.397,E2 -9159.397} C_VEL
LIN {X 0,Y 439.401,Z 203.053,A -85,B 0,C 180,E1 -9162.308,E2 -9162.308} C_VEL
LIN {X 0,Y 439.444,Z 203.054,A -85,B 0,C 180,E1 -9165.174,E2 -9165.174} C_VEL
LIN {X 0,Y 439.48,Z 203.034,A -85,B 0,C 180,E1 -9168.001,E2 -9168.001} C_VEL
LIN {X 0,Y 439.501,Z 203.047,A -85,B 0,C 180,E1 -9171.725,E2 -9171.725} C_VEL
LIN {X 0,Y 439.611,Z 203.03,A -85,B 0,C 180,E1 -9174.496,E2 -9174.496} C_VEL
LIN {X 0,Y 439.631,Z 203.013,A -85,B 0,C 180,E1 -9178.168,E2 -9178.168} C_VEL
LIN {X 0,Y 439.759,Z 203.013,A -85,B 0,C 180,E1 -9180,E2 -9180} C_VEL
LIN {X 0,Y 439.636,Z 203.03,A -85,B 0,C 180,E1 -9182.749,E2 -9182.749} C_VEL
LIN {X 0,Y 439.614,Z 203.032,A -85,B 0,C 180,E1 -9186.425,E2 -9186.425} C_VEL
LIN {X 0,Y 439.495,Z 203.048,A -85,B 0,C 180,E1 -9189.202,E2 -9189.202} C_VEL
LIN {X 0,Y 439.463,Z 203.045,A -85,B 0,C 180,E1 -9192.938,E2 -9192.938} C_VEL
LIN {X 0,Y 439.445,Z 203.054,A -85,B 0,C 180,E1 -9196.349,E2 -9196.349} C_VEL
LIN {X 0,Y 439.4,Z 203.05,A -85,B 0,C 180,E1 -9199.626,E2 -9199.626} C_VEL
LIN {X 0,Y 439.363,Z 203.065,A -85,B 0,C 180,E1 -9202.575,E2 -9202.575} C_VEL
LIN {X 0,Y 439.402,Z 203.052,A -85,B 0,C 180,E1 -9205.585,E2 -9205.585} C_VEL
LIN {X 0,Y 439.423,Z 203.058,A -85,B 0,C 180,E1 -9208.673,E2 -9208.673} C_VEL
LIN {X 0,Y 439.372,Z 203.057,A -85,B 0,C 180,E1 -9211.86,E2 -9211.86} C_VEL
LIN {X 0,Y 439.399,Z 203.063,A -85,B 0,C 180,E1 -9215.156,E2 -9215.156} C_VEL
LIN {X 0,Y 439.388,Z 203.054,A -85,B 0,C 180,E1 -9218.594,E2 -9218.594} C_VEL
LIN {X 0,Y 439.386,Z 203.066,A -85,B 0,C 180,E1 -9221.257,E2 -9221.257} C_VEL
LIN {X 0,Y 439.397,Z 203.056,A -85,B 0,C 180,E1 -9224.73,E2 -9224.73} C_VEL
LIN {X 0,Y 439.394,Z 203.06,A -85,B 0,C 180,E1 -9227.796,E2 -9227.796} C_VEL
LIN {X 0,Y 439.393,Z 203.061,A -85,B 0,C 180,E1 -9230.224,E2 -9230.224} C_VEL
LIN {X 0,Y 439.372,Z 203.059,A -85,B 0,C 180,E1 -9233.713,E2 -9233.713} C_VEL
LIN {X 0,Y 439.372,Z 203.07,A -85,B 0,C 180,E1 -9237.054,E2 -9237.054} C_VEL
LIN {X 0,Y 439.381,Z 203.064,A -85,B 0,C 180,E1 -9240.274,E2 -9240.274} C_VEL
LIN {X 0,Y 439.428,Z 203.058,A -85,B 0,C 180,E1 -9243.396,E2 -9243.396} C_VEL
LIN {X 0,Y 439.385,Z 203.058,A -85,B 0,C 180,E1 -9246.43,E2 -9246.43} C_VEL
LIN {X 0,Y 439.387,Z 203.057,A -85,B 0,C 180,E1 -9249.397,E2 -9249.397} C_VEL
LIN {X 0,Y 439.425,Z 203.053,A -85,B 0,C 180,E1 -9252.309,E2 -9252.309} C_VEL
LIN {X 0,Y 439.447,Z 203.047,A -85,B 0,C 180,E1 -9255.174,E2 -9255.174} C_VEL
LIN {X 0,Y 439.483,Z 203.053,A -85,B 0,C 180,E1 -9258.001,E2 -9258.001} C_VEL
LIN {X 0,Y 439.533,Z 203.049,A -85,B 0,C 180,E1 -9261.726,E2 -9261.726} C_VEL
LIN {X 0,Y 439.6,Z 203.175,A -85,B 0,C 180,E1 -9263.603,E2 -9263.603} C_VEL
LIN {X 0,Y 441.6,Z 209.772,A -85,B 0,C 180,E1 -9264.639,E2 -9264.639} C_VEL
LIN {X 0,Y 452.077,Z 231.119,A -85,B 0,C 180,E1 -9265.823,E2 -9265.823} C_VEL
LIN {X 0,Y 455.171,Z 237.87,A -85,B 0,C 180,E1 -9266.168,E2 -9266.168} C_VEL
LIN {X 0,Y 454.958,Z 252.973,A -85,B 0,C 180,E1 -9266.427,E2 -9266.427} C_VEL
LIN {X 0,Y 454.293,Z 258.817,A -85,B 0,C 180,E1 -9266.486,E2 -9266.486} C_VEL
LIN {X 0,Y 448.912,Z 277.902,A -85,B 0,C 180,E1 -9266.454,E2 -9266.454} C_VEL
LIN {X 0,Y 448.117,Z 283.754,A -85,B 0,C 180,E1 -9266.504,E2 -9266.504} C_VEL
LIN {X 0,Y 445.561,Z 415.849,A -85,B 0,C 180,E1 -9268.757,E2 -9268.757} C_VEL
LIN {X 0,Y 444.819,Z 432.937,A -85,B 0,C 180,E1 -9269.236,E2 -9269.236} C_VEL
LIN {X 0,Y 443.917,Z 448.065,A -85,B 0,C 180,E1 -9269.83,E2 -9269.83} C_VEL
LIN {X 0,Y 442.884,Z 463.137,A -85,B 0,C 180,E1 -9270.592,E2 -9270.592} C_VEL
LIN {X 0,Y 441.7,Z 477.374,A -85,B 0,C 180,E1 -9271.481,E2 -9271.481} C_VEL
LIN {X 0,Y 440.26,Z 492.39,A -85,B 0,C 180,E1 -9272.63,E2 -9272.63} C_VEL
LIN {X 0,Y 438.83,Z 506.192,A -85,B 0,C 180,E1 -9273.903,E2 -9273.903} C_VEL
LIN {X 0,Y 437.389,Z 519.518,A -85,B 0,C 180,E1 -9275.364,E2 -9275.364} C_VEL
LIN {X 0,Y 436.058,Z 531.677,A -85,B 0,C 180,E1 -9276.942,E2 -9276.942} C_VEL
LIN {X 0,Y 434.868,Z 542.388,A -85,B 0,C 180,E1 -9278.576,E2 -9278.576} C_VEL
LIN {X 0,Y 433.884,Z 551.737,A -85,B 0,C 180,E1 -9280.263,E2 -9280.263} C_VEL
LIN {X 0,Y 432.98,Z 560.761,A -85,B 0,C 180,E1 -9282.181,E2 -9282.181} C_VEL
LIN {X 0,Y 432.303,Z 568.346,A -85,B 0,C 180,E1 -9284.114,E2 -9284.114} C_VEL
LIN {X 0,Y 431.752,Z 574.95,A -85,B 0,C 180,E1 -9286.18,E2 -9286.18} C_VEL
LIN {X 0,Y 431.483,Z 579.611,A -85,B 0,C 180,E1 -9288.027,E2 -9288.027} C_VEL
LIN {X 0,Y 431.231,Z 583.55,A -85,B 0,C 180,E1 -9290.013,E2 -9290.013} C_VEL
LIN {X 0,Y 431.084,Z 586.324,A -85,B 0,C 180,E1 -9292.022,E2 -9292.022} C_VEL
LIN {X 0,Y 431.003,Z 587.998,A -85,B 0,C 180,E1 -9294.057,E2 -9294.057} C_VEL
LIN {X 0,Y 430.999,Z 588.573,A -85,B 0,C 180,E1 -9296.254,E2 -9296.254} C_VEL
LIN {X 0,Y 431.038,Z 587.905,A -85,B 0,C 180,E1 -9298.303,E2 -9298.303} C_VEL
LIN {X 0,Y 431.131,Z 586.076,A -85,B 0,C 180,E1 -9300.353,E2 -9300.353} C_VEL
LIN {X 0,Y 431.31,Z 582.891,A -85,B 0,C 180,E1 -9302.528,E2 -9302.528} C_VEL
LIN {X 0,Y 431.666,Z 578.249,A -85,B 0,C 180,E1 -9304.738,E2 -9304.738} C_VEL
LIN {X 0,Y 431.925,Z 573.618,A -85,B 0,C 180,E1 -9306.434,E2 -9306.434} C_VEL
LIN {X 0,Y 432.435,Z 566.947,A -85,B 0,C 180,E1 -9308.447,E2 -9308.447} C_VEL
LIN {X 0,Y 433.189,Z 558.789,A -85,B 0,C 180,E1 -9310.462,E2 -9310.462} C_VEL
LIN {X 0,Y 434.303,Z 548.563,A -85,B 0,C 180,E1 -9312.532,E2 -9312.532} C_VEL
LIN {X 0,Y 435.395,Z 538.322,A -85,B 0,C 180,E1 -9314.262,E2 -9314.262} C_VEL
LIN {X 0,Y 436.608,Z 528.016,A -85,B 0,C 180,E1 -9315.749,E2 -9315.749} C_VEL
LIN {X 0,Y 437.996,Z 516.101,A -85,B 0,C 180,E1 -9317.23,E2 -9317.23} C_VEL
LIN {X 0,Y 439.36,Z 503.314,A -85,B 0,C 180,E1 -9318.579,E2 -9318.579} C_VEL
LIN {X 0,Y 440.84,Z 489.607,A -85,B 0,C 180,E1 -9319.789,E2 -9319.789} C_VEL
LIN {X 0,Y 442.241,Z 474.339,A -85,B 0,C 180,E1 -9320.914,E2 -9320.914} C_VEL
LIN {X 0,Y 443.53,Z 458.93,A -85,B 0,C 180,E1 -9321.831,E2 -9321.831} C_VEL
LIN {X 0,Y 444.614,Z 442.64,A -85,B 0,C 180,E1 -9322.596,E2 -9322.596} C_VEL
LIN {X 0,Y 445.531,Z 426.032,A -85,B 0,C 180,E1 -9323.171,E2 -9323.171} C_VEL
LIN {X 0,Y 446.127,Z 408.57,A -85,B 0,C 180,E1 -9323.572,E2 -9323.572} C_VEL
LIN {X 0,Y 449.54,Z 241.481,A -85,B 0,C 180,E1 -9326.424,E2 -9326.424} C_VEL
LIN {X 0,Y 449.127,Z 239.714,A -85,B 0,C 180,E1 -9326.49,E2 -9326.49} C_VEL
LIN {X 0,Y 440.004,Z 220.957,A -85,B 0,C 180,E1 -9327.591,E2 -9327.591} C_VEL
LIN {X 0,Y 434.447,Z 210.606,A -85,B 0,C 180,E1 -9328.281,E2 -9328.281} C_VEL
LIN {X 0,Y 432.326,Z 203.946,A -85,B 0,C 180,E1 -9329.463,E2 -9329.463} C_VEL
LIN {X 0,Y 432.336,Z 203.946,A -85,B 0,C 180,E1 -9331.874,E2 -9331.874} C_VEL
LIN {X 0,Y 432.316,Z 203.944,A -85,B 0,C 180,E1 -9334.997,E2 -9334.997} C_VEL
LIN {X 0,Y 432.35,Z 203.936,A -85,B 0,C 180,E1 -9338.045,E2 -9338.045} C_VEL
LIN {X 0,Y 432.377,Z 203.935,A -85,B 0,C 180,E1 -9341.029,E2 -9341.029} C_VEL
LIN {X 0,Y 432.423,Z 203.927,A -85,B 0,C 180,E1 -9343.961,E2 -9343.961} C_VEL
LIN {X 0,Y 432.452,Z 203.92,A -85,B 0,C 180,E1 -9347.803,E2 -9347.803} C_VEL
LIN {X 0,Y 432.457,Z 203.926,A -85,B 0,C 180,E1 -9351.59,E2 -9351.59} C_VEL
LIN {X 0,Y 432.584,Z 203.915,A -85,B 0,C 180,E1 -9354.406,E2 -9354.406} C_VEL
LIN {X 0,Y 432.597,Z 203.911,A -85,B 0,C 180,E1 -9358.138,E2 -9358.138} C_VEL
LIN {X 0,Y 432.726,Z 203.897,A -85,B 0,C 180,E1 -9360,E2 -9360} C_VEL
LIN {X 0,Y 432.585,Z 203.909,A -85,B 0,C 180,E1 -9362.794,E2 -9362.794} C_VEL
LIN {X 0,Y 432.565,Z 203.916,A -85,B 0,C 180,E1 -9366.53,E2 -9366.53} C_VEL
LIN {X 0,Y 432.436,Z 203.929,A -85,B 0,C 180,E1 -9369.353,E2 -9369.353} C_VEL
LIN {X 0,Y 432.424,Z 203.93,A -85,B 0,C 180,E1 -9372.804,E2 -9372.804} C_VEL
LIN {X 0,Y 432.406,Z 203.932,A -85,B 0,C 180,E1 -9376.479,E2 -9376.479} C_VEL
LIN {X 0,Y 432.333,Z 203.947,A -85,B 0,C 180,E1 -9379.961,E2 -9379.961} C_VEL
LIN {X 0,Y 432.314,Z 203.945,A -85,B 0,C 180,E1 -9382.964,E2 -9382.964} C_VEL
LIN {X 0,Y 432.359,Z 203.939,A -85,B 0,C 180,E1 -9386.033,E2 -9386.033} C_VEL
LIN {X 0,Y 432.337,Z 203.943,A -85,B 0,C 180,E1 -9389.188,E2 -9389.188} C_VEL
LIN {X 0,Y 432.317,Z 203.946,A -85,B 0,C 180,E1 -9392.443,E2 -9392.443} C_VEL
LIN {X 0,Y 432.338,Z 203.946,A -85,B 0,C 180,E1 -9395.632,E2 -9395.632} C_VEL
LIN {X 0,Y 432.345,Z 203.949,A -85,B 0,C 180,E1 -9399.343,E2 -9399.343} C_VEL
LIN {X 0,Y 432.328,Z 203.948,A -85,B 0,C 180,E1 -9401.798,E2 -9401.798} C_VEL
LIN {X 0,Y 432.329,Z 203.948,A -85,B 0,C 180,E1 -9404.348,E2 -9404.348} C_VEL
LIN {X 0,Y 432.316,Z 203.951,A -85,B 0,C 180,E1 -9407.016,E2 -9407.016} C_VEL
LIN {X 0,Y 432.329,Z 203.946,A -85,B 0,C 180,E1 -9409.821,E2 -9409.821} C_VEL
LIN {X 0,Y 432.302,Z 203.949,A -85,B 0,C 180,E1 -9413.022,E2 -9413.022} C_VEL
LIN {X 0,Y 432.334,Z 204.055,A -85,B 0,C 180,E1 -9414.183,E2 -9414.183} C_VEL
LIN {X 0,Y 437.513,Z 219.467,A -85,B 0,C 180,E1 -9416.647,E2 -9416.647} C_VEL
LIN {X 0,Y 440.972,Z 230.764,A -85,B 0,C 180,E1 -9418.321,E2 -9418.321} C_VEL
LIN {X 0,Y 445.426,Z 240.341,A -85,B 0,C 180,E1 -9418.867,E2 -9418.867} C_VEL
LIN {X 0,Y 449.206,Z 262.901,A -85,B 0,C 180,E1 -9419.592,E2 -9419.592} C_VEL
LIN {X 0,Y 445.67,Z 438.028,A -85,B 0,C 180,E1 -9422.596,E2 -9422.596} C_VEL
LIN {X 0,Y 444.809,Z 453.844,A -85,B 0,C 180,E1 -9423.016,E2 -9423.016} C_VEL
LIN {X 0,Y 443.858,Z 469.796,A -85,B 0,C 180,E1 -9423.62,E2 -9423.62} C_VEL
LIN {X 0,Y 442.649,Z 485.067,A -85,B 0,C 180,E1 -9424.365,E2 -9424.365} C_VEL
LIN {X 0,Y 441.355,Z 500.093,A -85,B 0,C 180,E1 -9425.294,E2 -9425.294} C_VEL
LIN {X 0,Y 439.908,Z 513.992,A -85,B 0,C 180,E1 -9426.335,E2 -9426.335} C_VEL
LIN {X 0,Y 438.412,Z 528.331,A -85,B 0,C 180,E1 -9427.622,E2 -9427.622} C_VEL
LIN {X 0,Y 436.992,Z 541.268,A -85,B 0,C 180,E1 -9428.998,E2 -9428.998} C_VEL
LIN {X 0,Y 435.712,Z 552.838,A -85,B 0,C 180,E1 -9430.447,E2 -9430.447} C_VEL
LIN {X 0,Y 434.451,Z 564.112,A -85,B 0,C 180,E1 -9432.1,E2 -9432.1} C_VEL
LIN {X 0,Y 433.486,Z 575.046,A -85,B 0,C 180,E1 -9434.002,E2 -9434.002} C_VEL
LIN {X 0,Y 432.563,Z 584.237,A -85,B 0,C 180,E1 -9435.895,E2 -9435.895} C_VEL
LIN {X 0,Y 432.045,Z 591.941,A -85,B 0,C 180,E1 -9437.792,E2 -9437.792} C_VEL
LIN {X 0,Y 431.485,Z 599.68,A -85,B 0,C 180,E1 -9440.153,E2 -9440.153} C_VEL
LIN {X 0,Y 431.307,Z 605.575,A -85,B 0,C 180,E1 -9442.51,E2 -9442.51} C_VEL
LIN {X 0,Y 431.22,Z 609.025,A -85,B 0,C 180,E1 -9444.389,E2 -9444.389} C_VEL
LIN {X 0,Y 431.138,Z 611.534,A -85,B 0,C 180,E1 -9446.262,E2 -9446.262} C_VEL
LIN {X 0,Y 431.212,Z 612.955,A -85,B 0,C 180,E1 -9448.132,E2 -9448.132} C_VEL
LIN {X 0,Y 431.163,Z 613.492,A -85,B 0,C 180,E1 -9450,E2 -9450} C_VEL
LIN {X 0,Y 431.212,Z 612.965,A -85,B 0,C 180,E1 -9451.868,E2 -9451.868} C_VEL
LIN {X 0,Y 431.138,Z 611.551,A -85,B 0,C 180,E1 -9453.739,E2 -9453.739} C_VEL
LIN {X 0,Y 431.22,Z 609.052,A -85,B 0,C 180,E1 -9455.612,E2 -9455.612} C_VEL
LIN {X 0,Y 431.308,Z 605.604,A -85,B 0,C 180,E1 -9457.49,E2 -9457.49} C_VEL
LIN {X 0,Y 431.488,Z 599.71,A -85,B 0,C 180,E1 -9459.847,E2 -9459.847} C_VEL
LIN {X 0,Y 431.911,Z 593.632,A -85,B 0,C 180,E1 -9461.736,E2 -9461.736} C_VEL
LIN {X 0,Y 432.408,Z 586.284,A -85,B 0,C 180,E1 -9463.631,E2 -9463.631} C_VEL
LIN {X 0,Y 433.174,Z 577.506,A -85,B 0,C 180,E1 -9465.528,E2 -9465.528} C_VEL
LIN {X 0,Y 434.176,Z 567.096,A -85,B 0,C 180,E1 -9467.412,E2 -9467.412} C_VEL
LIN {X 0,Y 435.313,Z 556.105,A -85,B 0,C 180,E1 -9469.083,E2 -9469.083} C_VEL
LIN {X 0,Y 436.682,Z 543.286,A -85,B 0,C 180,E1 -9470.736,E2 -9470.736} C_VEL
LIN {X 0,Y 438.064,Z 530.326,A -85,B 0,C 180,E1 -9472.149,E2 -9472.149} C_VEL
LIN {X 0,Y 439.543,Z 516.305,A -85,B 0,C 180,E1 -9473.437,E2 -9473.437} C_VEL
LIN {X 0,Y 441.082,Z 500.917,A -85,B 0,C 180,E1 -9474.605,E2 -9474.605} C_VEL
LIN {X 0,Y 442.501,Z 485.004,A -85,B 0,C 180,E1 -9475.582,E2 -9475.582} C_VEL
LIN {X 0,Y 443.642,Z 469.515,A -85,B 0,C 180,E1 -9476.331,E2 -9476.331} C_VEL
LIN {X 0,Y 444.518,Z 453.158,A -85,B 0,C 180,E1 -9476.94,E2 -9476.94} C_VEL
LIN {X 0,Y 445.399,Z 436.317,A -85,B 0,C 180,E1 -9477.363,E2 -9477.363} C_VEL
LIN {X 0,Y 448.799,Z 263.208,A -85,B 0,C 180,E1 -9480.298,E2 -9480.298} C_VEL
LIN {X 0,Y 444.569,Z 239.189,A -85,B 0,C 180,E1 -9481.055,E2 -9481.055} C_VEL
LIN {X 0,Y 440.933,Z 231.28,A -85,B 0,C 180,E1 -9481.491,E2 -9481.491} C_VEL
LIN {X 0,Y 435.325,Z 213.014,A -85,B 0,C 180,E1 -9484.168,E2 -9484.168} C_VEL
LIN {X 0,Y 432.338,Z 203.942,A -85,B 0,C 180,E1 -9485.583,E2 -9485.583} C_VEL
LIN {X 0,Y 432.336,Z 203.947,A -85,B 0,C 180,E1 -9488.714,E2 -9488.714} C_VEL
LIN {X 0,Y 432.322,Z 203.945,A -85,B 0,C 180,E1 -9491.798,E2 -9491.798} C_VEL
LIN {X 0,Y 432.331,Z 203.944,A -85,B 0,C 180,E1 -9494.347,E2 -9494.347} C_VEL
LIN {X 0,Y 432.314,Z 203.947,A -85,B 0,C 180,E1 -9497.016,E2 -9497.016} C_VEL
LIN {X 0,Y 432.31,Z 203.941,A -85,B 0,C 180,E1 -9499.824,E2 -9499.824} C_VEL
LIN {X 0,Y 432.303,Z 203.94,A -85,B 0,C 180,E1 -9503.022,E2 -9503.022} C_VEL
LIN {X 0,Y 432.355,Z 203.94,A -85,B 0,C 180,E1 -9505.997,E2 -9505.997} C_VEL
LIN {X 0,Y 432.344,Z 203.938,A -85,B 0,C 180,E1 -9509.49,E2 -9509.49} C_VEL
LIN {X 0,Y 432.387,Z 203.927,A -85,B 0,C 180,E1 -9512.928,E2 -9512.928} C_VEL
LIN {X 0,Y 432.365,Z 203.935,A -85,B 0,C 180,E1 -9516.023,E2 -9516.023} C_VEL
LIN {X 0,Y 432.346,Z 203.933,A -85,B 0,C 180,E1 -9519.046,E2 -9519.046} C_VEL
LIN {X 0,Y 432.357,Z 203.928,A -85,B 0,C 180,E1 -9522.01,E2 -9522.01} C_VEL
LIN {X 0,Y 432.392,Z 203.935,A -85,B 0,C 180,E1 -9524.926,E2 -9524.926} C_VEL
LIN {X 0,Y 432.456,Z 203.909,A -85,B 0,C 180,E1 -9527.803,E2 -9527.803} C_VEL
LIN {X 0,Y 432.461,Z 203.924,A -85,B 0,C 180,E1 -9531.59,E2 -9531.59} C_VEL
LIN {X 0,Y 432.588,Z 203.905,A -85,B 0,C 180,E1 -9534.406,E2 -9534.406} C_VEL
LIN {X 0,Y 432.601,Z 203.887,A -85,B 0,C 180,E1 -9538.138,E2 -9538.138} C_VEL
LIN {X 0,Y 432.728,Z 203.888,A -85,B 0,C 180,E1 -9540,E2 -9540} C_VEL
LIN {X 0,Y 432.588,Z 203.908,A -85,B 0,C 180,E1 -9542.794,E2 -9542.794} C_VEL
LIN {X 0,Y 432.569,Z 203.911,A -85,B 0,C 180,E1 -9546.53,E2 -9546.53} C_VEL
LIN {X 0,Y 432.438,Z 203.927,A -85,B 0,C 180,E1 -9549.353,E2 -9549.353} C_VEL
LIN {X 0,Y 432.428,Z 203.922,A -85,B 0,C 180,E1 -9552.803,E2 -9552.803} C_VEL
LIN {X 0,Y 432.41,Z 203.929,A -85,B 0,C 180,E1 -9556.479,E2 -9556.479} C_VEL
LIN {X 0,Y 432.336,Z 203.934,A -85,B 0,C 180,E1 -9559.96,E2 -9559.96} C_VEL
LIN {X 0,Y 432.317,Z 203.942,A -85,B 0,C 180,E1 -9562.964,E2 -9562.964} C_VEL
LIN {X 0,Y 432.362,Z 203.93,A -85,B 0,C 180,E1 -9566.032,E2 -9566.032} C_VEL
LIN {X 0,Y 432.35,Z 203.94,A -85,B 0,C 180,E1 -9569.187,E2 -9569.187} C_VEL
LIN {X 0,Y 432.323,Z 203.935,A -85,B 0,C 180,E1 -9572.293,E2 -9572.293} C_VEL
LIN {X 0,Y 432.339,Z 203.94,A -85,B 0,C 180,E1 -9574.677,E2 -9574.677} C_VEL
LIN {X 0,Y 432.345,Z 203.932,A -85,B 0,C 180,E1 -9578.149,E2 -9578.149} C_VEL
LIN {X 0,Y 432.331,Z 203.946,A -85,B 0,C 180,E1 -9581.602,E2 -9581.602} C_VEL
LIN {X 0,Y 432.331,Z 203.936,A -85,B 0,C 180,E1 -9584.347,E2 -9584.347} C_VEL
LIN {X 0,Y 432.318,Z 203.946,A -85,B 0,C 180,E1 -9587.016,E2 -9587.016} C_VEL
LIN {X 0,Y 432.331,Z 203.942,A -85,B 0,C 180,E1 -9589.821,E2 -9589.821} C_VEL
LIN {X 0,Y 432.305,Z 203.945,A -85,B 0,C 180,E1 -9593.022,E2 -9593.022} C_VEL
LIN {X 0,Y 432.358,Z 203.94,A -85,B 0,C 180,E1 -9595.997,E2 -9595.997} C_VEL
LIN {X 0,Y 432.346,Z 203.94,A -85,B 0,C 180,E1 -9599.49,E2 -9599.49} C_VEL
LIN {X 0,Y 432.39,Z 203.931,A -85,B 0,C 180,E1 -9602.928,E2 -9602.928} C_VEL
LIN {X 0,Y 432.37,Z 203.932,A -85,B 0,C 180,E1 -9606.023,E2 -9606.023} C_VEL
LIN {X 0,Y 432.349,Z 203.938,A -85,B 0,C 180,E1 -9609.046,E2 -9609.046} C_VEL
LIN {X 0,Y 432.373,Z 203.927,A -85,B 0,C 180,E1 -9612.011,E2 -9612.011} C_VEL
LIN {X 0,Y 432.395,Z 203.929,A -85,B 0,C 180,E1 -9614.926,E2 -9614.926} C_VEL
LIN {X 0,Y 432.459,Z 203.929,A -85,B 0,C 180,E1 -9617.803,E2 -9617.803} C_VEL
LIN {X 0,Y 432.482,Z 203.927,A -85,B 0,C 180,E1 -9621.59,E2 -9621.59} C_VEL
LIN {X 0,Y 432.527,Z 203.937,A -85,B 0,C 180,E1 -9623.104,E2 -9623.104} C_VEL
LIN {X 0,Y 434.455,Z 210.056,A -85,B 0,C 180,E1 -9624.081,E2 -9624.081} C_VEL
LIN {X 0,Y 446.582,Z 234.798,A -85,B 0,C 180,E1 -9625.487,E2 -9625.487} C_VEL
LIN {X 0,Y 448.952,Z 239.977,A -85,B 0,C 180,E1 -9625.758,E2 -9625.758} C_VEL
LIN {X 0,Y 448.117,Z 283.754,A -85,B 0,C 180,E1 -9626.504,E2 -9626.504} C_VEL
LIN {X 0,Y 447.326,Z 289.605,A -85,B 0,C 180,E1 -9626.556,E2 -9626.556} C_VEL
LIN {X 0,Y 441.926,Z 308.686,A -85,B 0,C 180,E1 -9626.524,E2 -9626.524} C_VEL
LIN {X 0,Y 441.216,Z 314.533,A -85,B 0,C 180,E1 -9626.582,E2 -9626.582} C_VEL
LIN {X 0,Y 439.227,Z 415.75,A -85,B 0,C 180,E1 -9628.338,E2 -9628.338} C_VEL
LIN {X 0,Y 438.477,Z 432.914,A -85,B 0,C 180,E1 -9628.823,E2 -9628.823} C_VEL
LIN {X 0,Y 437.516,Z 448.137,A -85,B 0,C 180,E1 -9629.425,E2 -9629.425} C_VEL
LIN {X 0,Y 436.376,Z 464.113,A -85,B 0,C 180,E1 -9630.249,E2 -9630.249} C_VEL
LIN {X 0,Y 435.137,Z 478.333,A -85,B 0,C 180,E1 -9631.157,E2 -9631.157} C_VEL
LIN {X 0,Y 433.621,Z 493.237,A -85,B 0,C 180,E1 -9632.322,E2 -9632.322} C_VEL
LIN {X 0,Y 432.132,Z 506.93,A -85,B 0,C 180,E1 -9633.613,E2 -9633.613} C_VEL
LIN {X 0,Y 430.724,Z 519.323,A -85,B 0,C 180,E1 -9634.993,E2 -9634.993} C_VEL
LIN {X 0,Y 429.316,Z 531.453,A -85,B 0,C 180,E1 -9636.58,E2 -9636.58} C_VEL
LIN {X 0,Y 428.021,Z 542.341,A -85,B 0,C 180,E1 -9638.26,E2 -9638.26} C_VEL
LIN {X 0,Y 426.97,Z 551.628,A -85,B 0,C 180,E1 -9639.952,E2 -9639.952} C_VEL
LIN {X 0,Y 426.036,Z 560.701,A -85,B 0,C 180,E1 -9641.9,E2 -9641.9} C_VEL
LIN {X 0,Y 425.318,Z 568.338,A -85,B 0,C 180,E1 -9643.862,E2 -9643.862} C_VEL
LIN {X 0,Y 424.739,Z 574.547,A -85,B 0,C 180,E1 -9645.82,E2 -9645.82} C_VEL
LIN {X 0,Y 424.434,Z 579.673,A -85,B 0,C 180,E1 -9647.838,E2 -9647.838} C_VEL
LIN {X 0,Y 424.223,Z 582.741,A -85,B 0,C 180,E1 -9649.349,E2 -9649.349} C_VEL
LIN {X 0,Y 424.036,Z 585.848,A -85,B 0,C 180,E1 -9651.384,E2 -9651.384} C_VEL
LIN {X 0,Y 423.916,Z 587.879,A -85,B 0,C 180,E1 -9653.446,E2 -9653.446} C_VEL
LIN {X 0,Y 423.869,Z 588.719,A -85,B 0,C 180,E1 -9655.536,E2 -9655.536} C_VEL
LIN {X 0,Y 423.909,Z 588.449,A -85,B 0,C 180,E1 -9657.659,E2 -9657.659} C_VEL
LIN {X 0,Y 424,Z 586.98,A -85,B 0,C 180,E1 -9659.818,E2 -9659.818} C_VEL
LIN {X 0,Y 424.194,Z 584.134,A -85,B 0,C 180,E1 -9662.016,E2 -9662.016} C_VEL
LIN {X 0,Y 424.496,Z 579.879,A -85,B 0,C 180,E1 -9664.256,E2 -9664.256} C_VEL
LIN {X 0,Y 424.817,Z 575.18,A -85,B 0,C 180,E1 -9666.153,E2 -9666.153} C_VEL
LIN {X 0,Y 425.351,Z 568.51,A -85,B 0,C 180,E1 -9668.286,E2 -9668.286} C_VEL
LIN {X 0,Y 426.124,Z 560.482,A -85,B 0,C 180,E1 -9670.357,E2 -9670.357} C_VEL
LIN {X 0,Y 427.049,Z 551.798,A -85,B 0,C 180,E1 -9672.22,E2 -9672.22} C_VEL
LIN {X 0,Y 428.159,Z 542.362,A -85,B 0,C 180,E1 -9673.943,E2 -9673.943} C_VEL
LIN {X 0,Y 429.452,Z 531.865,A -85,B 0,C 180,E1 -9675.571,E2 -9675.571} C_VEL
LIN {X 0,Y 430.964,Z 519.42,A -85,B 0,C 180,E1 -9677.208,E2 -9677.208} C_VEL
LIN {X 0,Y 432.378,Z 507.278,A -85,B 0,C 180,E1 -9678.566,E2 -9678.566} C_VEL
LIN {X 0,Y 433.833,Z 494.728,A -85,B 0,C 180,E1 -9679.765,E2 -9679.765} C_VEL
LIN {X 0,Y 435.387,Z 479.38,A -85,B 0,C 180,E1 -9680.984,E2 -9680.984} C_VEL
LIN {X 0,Y 436.775,Z 464.384,A -85,B 0,C 180,E1 -9681.948,E2 -9681.948} C_VEL
LIN {X 0,Y 437.878,Z 449.217,A -85,B 0,C 180,E1 -9682.738,E2 -9682.738} C_VEL
LIN {X 0,Y 438.881,Z 433.299,A -85,B 0,C 180,E1 -9683.374,E2 -9683.374} C_VEL
LIN {X 0,Y 439.677,Z 416.789,A -85,B 0,C 180,E1 -9683.844,E2 -9683.844} C_VEL
LIN {X 0,Y 443.452,Z 242.73,A -85,B 0,C 180,E1 -9686.884,E2 -9686.884} C_VEL
LIN {X 0,Y 434.906,Z 225.124,A -85,B 0,C 180,E1 -9687.944,E2 -9687.944} C_VEL
LIN {X 0,Y 427.233,Z 210.862,A -85,B 0,C 180,E1 -9688.928,E2 -9688.928} C_VEL
LIN {X 0,Y 425.278,Z 204.827,A -85,B 0,C 180,E1 -9690.041,E2 -9690.041} C_VEL
LIN {X 0,Y 425.273,Z 204.821,A -85,B 0,C 180,E1 -9693.174,E2 -9693.174} C_VEL
LIN {X 0,Y 425.316,Z 204.815,A -85,B 0,C 180,E1 -9695.6,E2 -9695.6} C_VEL
LIN {X 0,Y 425.286,Z 204.82,A -85,B 0,C 180,E1 -9698.681,E2 -9698.681} C_VEL
LIN {X 0,Y 425.315,Z 204.817,A -85,B 0,C 180,E1 -9701.702,E2 -9701.702} C_VEL
LIN {X 0,Y 425.34,Z 204.809,A -85,B 0,C 180,E1 -9704.67,E2 -9704.67} C_VEL
LIN {X 0,Y 425.405,Z 204.799,A -85,B 0,C 180,E1 -9707.598,E2 -9707.598} C_VEL
LIN {X 0,Y 425.401,Z 204.805,A -85,B 0,C 180,E1 -9711.449,E2 -9711.449} C_VEL
LIN {X 0,Y 425.539,Z 204.792,A -85,B 0,C 180,E1 -9714.313,E2 -9714.313} C_VEL
LIN {X 0,Y 425.566,Z 204.786,A -85,B 0,C 180,E1 -9718.107,E2 -9718.107} C_VEL
LIN {X 0,Y 425.696,Z 204.773,A -85,B 0,C 180,E1 -9720,E2 -9720} C_VEL
LIN {X 0,Y 425.539,Z 204.786,A -85,B 0,C 180,E1 -9722.84,E2 -9722.84} C_VEL
LIN {X 0,Y 425.523,Z 204.793,A -85,B 0,C 180,E1 -9726.639,E2 -9726.639} C_VEL
LIN {X 0,Y 425.395,Z 204.807,A -85,B 0,C 180,E1 -9729.509,E2 -9729.509} C_VEL
LIN {X 0,Y 425.387,Z 204.807,A -85,B 0,C 180,E1 -9732.904,E2 -9732.904} C_VEL
LIN {X 0,Y 425.355,Z 204.81,A -85,B 0,C 180,E1 -9736.605,E2 -9736.605} C_VEL
LIN {X 0,Y 425.322,Z 204.816,A -85,B 0,C 180,E1 -9739.636,E2 -9739.636} C_VEL
LIN {X 0,Y 425.301,Z 204.822,A -85,B 0,C 180,E1 -9743.365,E2 -9743.365} C_VEL
LIN {X 0,Y 425.343,Z 204.81,A -85,B 0,C 180,E1 -9746.845,E2 -9746.845} C_VEL
LIN {X 0,Y 425.285,Z 204.824,A -85,B 0,C 180,E1 -9749.72,E2 -9749.72} C_VEL
LIN {X 0,Y 425.276,Z 204.826,A -85,B 0,C 180,E1 -9753.048,E2 -9753.048} C_VEL
LIN {X 0,Y 425.277,Z 204.825,A -85,B 0,C 180,E1 -9755.929,E2 -9755.929} C_VEL
LIN {X 0,Y 425.292,Z 204.827,A -85,B 0,C 180,E1 -9759.044,E2 -9759.044} C_VEL
LIN {X 0,Y 425.27,Z 204.828,A -85,B 0,C 180,E1 -9762.653,E2 -9762.653} C_VEL
LIN {X 0,Y 425.257,Z 204.829,A -85,B 0,C 180,E1 -9766.045,E2 -9766.045} C_VEL
LIN {X 0,Y 425.269,Z 204.828,A -85,B 0,C 180,E1 -9768.622,E2 -9768.622} C_VEL
LIN {X 0,Y 425.302,Z 204.824,A -85,B 0,C 180,E1 -9771.103,E2 -9771.103} C_VEL
LIN {X 0,Y 425.309,Z 204.996,A -85,B 0,C 180,E1 -9773.618,E2 -9773.618} C_VEL
LIN {X 0,Y 430.88,Z 221.45,A -85,B 0,C 180,E1 -9776.32,E2 -9776.32} C_VEL
LIN {X 0,Y 433.677,Z 230.448,A -85,B 0,C 180,E1 -9777.695,E2 -9777.695} C_VEL
LIN {X 0,Y 439.651,Z 243.218,A -85,B 0,C 180,E1 -9778.455,E2 -9778.455} C_VEL
LIN {X 0,Y 443.123,Z 264.436,A -85,B 0,C 180,E1 -9779.145,E2 -9779.145} C_VEL
LIN {X 0,Y 439.377,Z 438.501,A -85,B 0,C 180,E1 -9782.176,E2 -9782.176} C_VEL
LIN {X 0,Y 438.441,Z 454.781,A -85,B 0,C 180,E1 -9782.623,E2 -9782.623} C_VEL
LIN {X 0,Y 437.497,Z 469.749,A -85,B 0,C 180,E1 -9783.206,E2 -9783.206} C_VEL
LIN {X 0,Y 436.213,Z 484.978,A -85,B 0,C 180,E1 -9783.958,E2 -9783.958} C_VEL
LIN {X 0,Y 434.853,Z 499.887,A -85,B 0,C 180,E1 -9784.892,E2 -9784.892} C_VEL
LIN {X 0,Y 433.349,Z 513.866,A -85,B 0,C 180,E1 -9785.954,E2 -9785.954} C_VEL
LIN {X 0,Y 431.786,Z 528.173,A -85,B 0,C 180,E1 -9787.259,E2 -9787.259} C_VEL
LIN {X 0,Y 430.381,Z 540.293,A -85,B 0,C 180,E1 -9788.558,E2 -9788.558} C_VEL
LIN {X 0,Y 428.918,Z 552.651,A -85,B 0,C 180,E1 -9790.124,E2 -9790.124} C_VEL
LIN {X 0,Y 427.611,Z 563.924,A -85,B 0,C 180,E1 -9791.804,E2 -9791.804} C_VEL
LIN {X 0,Y 426.639,Z 573.607,A -85,B 0,C 180,E1 -9793.492,E2 -9793.492} C_VEL
LIN {X 0,Y 425.698,Z 583.021,A -85,B 0,C 180,E1 -9795.418,E2 -9795.418} C_VEL
LIN {X 0,Y 424.993,Z 591.747,A -85,B 0,C 180,E1 -9797.586,E2 -9797.586} C_VEL
LIN {X 0,Y 424.428,Z 599.481,A -85,B 0,C 180,E1 -9799.988,E2 -9799.988} C_VEL
LIN {X 0,Y 424.225,Z 605.374,A -85,B 0,C 180,E1 -9802.384,E2 -9802.384} C_VEL
LIN {X 0,Y 424.14,Z 608.824,A -85,B 0,C 180,E1 -9804.295,E2 -9804.295} C_VEL
LIN {X 0,Y 424.05,Z 611.331,A -85,B 0,C 180,E1 -9806.199,E2 -9806.199} C_VEL
LIN {X 0,Y 424.136,Z 612.752,A -85,B 0,C 180,E1 -9808.101,E2 -9808.101} C_VEL
LIN {X 0,Y 424.08,Z 613.287,A -85,B 0,C 180,E1 -9810,E2 -9810} C_VEL
LIN {X 0,Y 424.137,Z 612.758,A -85,B 0,C 180,E1 -9811.899,E2 -9811.899} C_VEL
LIN {X 0,Y 424.05,Z 611.34,A -85,B 0,C 180,E1 -9813.801,E2 -9813.801} C_VEL
LIN {X 0,Y 424.224,Z 607.947,A -85,B 0,C 180,E1 -9816.28,E2 -9816.28} C_VEL
LIN {X 0,Y 424.274,Z 603.224,A -85,B 0,C 180,E1 -9818.574,E2 -9818.574} C_VEL
LIN {X 0,Y 424.533,Z 598.042,A -85,B 0,C 180,E1 -9820.492,E2 -9820.492} C_VEL
LIN {X 0,Y 425.008,Z 591.718,A -85,B 0,C 180,E1 -9822.414,E2 -9822.414} C_VEL
LIN {X 0,Y 425.657,Z 582.961,A -85,B 0,C 180,E1 -9824.584,E2 -9824.584} C_VEL
LIN {X 0,Y 426.627,Z 573.507,A -85,B 0,C 180,E1 -9826.509,E2 -9826.509} C_VEL
LIN {X 0,Y 427.602,Z 563.745,A -85,B 0,C 180,E1 -9828.197,E2 -9828.197} C_VEL
LIN {X 0,Y 428.875,Z 552.364,A -85,B 0,C 180,E1 -9829.879,E2 -9829.879} C_VEL
LIN {X 0,Y 430.328,Z 540.067,A -85,B 0,C 180,E1 -9831.424,E2 -9831.424} C_VEL
LIN {X 0,Y 431.866,Z 526.448,A -85,B 0,C 180,E1 -9832.863,E2 -9832.863} C_VEL
LIN {X 0,Y 433.258,Z 513.071,A -85,B 0,C 180,E1 -9834.052,E2 -9834.052} C_VEL
LIN {X 0,Y 434.691,Z 498.674,A -85,B 0,C 180,E1 -9835.124,E2 -9835.124} C_VEL
LIN {X 0,Y 436.167,Z 483.477,A -85,B 0,C 180,E1 -9836.045,E2 -9836.045} C_VEL
LIN {X 0,Y 437.357,Z 467.726,A -85,B 0,C 180,E1 -9836.804,E2 -9836.804} C_VEL
LIN {X 0,Y 438.219,Z 452.563,A -85,B 0,C 180,E1 -9837.36,E2 -9837.36} C_VEL
LIN {X 0,Y 439.083,Z 435.864,A -85,B 0,C 180,E1 -9837.782,E2 -9837.782} C_VEL
LIN {X 0,Y 442.565,Z 264.001,A -85,B 0,C 180,E1 -9840.739,E2 -9840.739} C_VEL
LIN {X 0,Y 438.749,Z 242.084,A -85,B 0,C 180,E1 -9841.442,E2 -9841.442} C_VEL
LIN {X 0,Y 433.616,Z 230.992,A -85,B 0,C 180,E1 -9842.075,E2 -9842.075} C_VEL
LIN {X 0,Y 427.992,Z 212.818,A -85,B 0,C 180,E1 -9844.811,E2 -9844.811} C_VEL
LIN {X 0,Y 425.285,Z 204.823,A -85,B 0,C 180,E1 -9846.095,E2 -9846.095} C_VEL
LIN {X 0,Y 425.279,Z 204.826,A -85,B 0,C 180,E1 -9849.041,E2 -9849.041} C_VEL
LIN {X 0,Y 425.28,Z 204.822,A -85,B 0,C 180,E1 -9851.957,E2 -9851.957} C_VEL
LIN {X 0,Y 425.282,Z 204.816,A -85,B 0,C 180,E1 -9855.283,E2 -9855.283} C_VEL
LIN {X 0,Y 425.262,Z 204.822,A -85,B 0,C 180,E1 -9858.62,E2 -9858.62} C_VEL
LIN {X 0,Y 425.289,Z 204.826,A -85,B 0,C 180,E1 -9861.1,E2 -9861.1} C_VEL
LIN {X 0,Y 425.295,Z 204.814,A -85,B 0,C 180,E1 -9864.664,E2 -9864.664} C_VEL
LIN {X 0,Y 425.261,Z 204.813,A -85,B 0,C 180,E1 -9868.073,E2 -9868.073} C_VEL
LIN {X 0,Y 425.328,Z 204.816,A -85,B 0,C 180,E1 -9871.368,E2 -9871.368} C_VEL
LIN {X 0,Y 425.351,Z 204.799,A -85,B 0,C 180,E1 -9873.505,E2 -9873.505} C_VEL
LIN {X 0,Y 425.302,Z 204.821,A -85,B 0,C 180,E1 -9876.635,E2 -9876.635} C_VEL
LIN {X 0,Y 425.325,Z 204.8,A -85,B 0,C 180,E1 -9880.365,E2 -9880.365} C_VEL
LIN {X 0,Y 425.385,Z 204.806,A -85,B 0,C 180,E1 -9883.688,E2 -9883.688} C_VEL
LIN {X 0,Y 425.409,Z 204.788,A -85,B 0,C 180,E1 -9887.598,E2 -9887.598} C_VEL
LIN {X 0,Y 425.405,Z 204.802,A -85,B 0,C 180,E1 -9891.449,E2 -9891.449} C_VEL
LIN {X 0,Y 425.543,Z 204.784,A -85,B 0,C 180,E1 -9894.313,E2 -9894.313} C_VEL
LIN {X 0,Y 425.57,Z 204.762,A -85,B 0,C 180,E1 -9898.107,E2 -9898.107} C_VEL
LIN {X 0,Y 425.698,Z 204.764,A -85,B 0,C 180,E1 -9900,E2 -9900} C_VEL
LIN {X 0,Y 425.542,Z 204.785,A -85,B 0,C 180,E1 -9902.84,E2 -9902.84} C_VEL
LIN {X 0,Y 425.526,Z 204.788,A -85,B 0,C 180,E1 -9906.651,E2 -9906.651} C_VEL
LIN {X 0,Y 425.397,Z 204.805,A -85,B 0,C 180,E1 -9909.509,E2 -9909.509} C_VEL
LIN {X 0,Y 425.391,Z 204.798,A -85,B 0,C 180,E1 -9912.904,E2 -9912.904} C_VEL
LIN {X 0,Y 425.359,Z 204.806,A -85,B 0,C 180,E1 -9916.605,E2 -9916.605} C_VEL
LIN {X 0,Y 425.326,Z 204.803,A -85,B 0,C 180,E1 -9919.636,E2 -9919.636} C_VEL
LIN {X 0,Y 425.305,Z 204.817,A -85,B 0,C 180,E1 -9923.365,E2 -9923.365} C_VEL
LIN {X 0,Y 425.346,Z 204.806,A -85,B 0,C 180,E1 -9926.844,E2 -9926.844} C_VEL
LIN {X 0,Y 425.316,Z 204.819,A -85,B 0,C 180,E1 -9929.717,E2 -9929.717} C_VEL
LIN {X 0,Y 425.28,Z 204.812,A -85,B 0,C 180,E1 -9933.048,E2 -9933.048} C_VEL
LIN {X 0,Y 425.282,Z 204.821,A -85,B 0,C 180,E1 -9935.929,E2 -9935.929} C_VEL
LIN {X 0,Y 425.301,Z 204.809,A -85,B 0,C 180,E1 -9939.044,E2 -9939.044} C_VEL
LIN {X 0,Y 425.272,Z 204.818,A -85,B 0,C 180,E1 -9942.653,E2 -9942.653} C_VEL
LIN {X 0,Y 425.259,Z 204.825,A -85,B 0,C 180,E1 -9946.044,E2 -9946.044} C_VEL
LIN {X 0,Y 425.272,Z 204.815,A -85,B 0,C 180,E1 -9948.621,E2 -9948.621} C_VEL
LIN {X 0,Y 425.295,Z 204.82,A -85,B 0,C 180,E1 -9951.101,E2 -9951.101} C_VEL
LIN {X 0,Y 425.298,Z 204.811,A -85,B 0,C 180,E1 -9954.664,E2 -9954.664} C_VEL
LIN {X 0,Y 425.264,Z 204.816,A -85,B 0,C 180,E1 -9958.073,E2 -9958.073} C_VEL
LIN {X 0,Y 425.33,Z 204.816,A -85,B 0,C 180,E1 -9961.368,E2 -9961.368} C_VEL
LIN {X 0,Y 425.294,Z 204.82,A -85,B 0,C 180,E1 -9964.555,E2 -9964.555} C_VEL
LIN {X 0,Y 425.287,Z 204.823,A -85,B 0,C 180,E1 -9967.661,E2 -9967.661} C_VEL
LIN {X 0,Y 425.36,Z 204.792,A -85,B 0,C 180,E1 -9970.704,E2 -9970.704} C_VEL
LIN {X 0,Y 425.387,Z 204.812,A -85,B 0,C 180,E1 -9973.688,E2 -9973.688} C_VEL
LIN {X 0,Y 425.412,Z 204.804,A -85,B 0,C 180,E1 -9977.598,E2 -9977.598} C_VEL
LIN {X 0,Y 425.436,Z 204.803,A -85,B 0,C 180,E1 -9981.45,E2 -9981.45} C_VEL
LIN {X 0,Y 425.485,Z 204.849,A -85,B 0,C 180,E1 -9982.612,E2 -9982.612} C_VEL
LIN {X 0,Y 427.204,Z 210.25,A -85,B 0,C 180,E1 -9983.493,E2 -9983.493} C_VEL
LIN {X 0,Y 440.753,Z 237.601,A -85,B 0,C 180,E1 -9985.101,E2 -9985.101} C_VEL
LIN {X 0,Y 442.706,Z 242.038,A -85,B 0,C 180,E1 -9985.333,E2 -9985.333} C_VEL
LIN {X 0,Y 441.216,Z 314.533,A -85,B 0,C 180,E1 -9986.582,E2 -9986.582} C_VEL
LIN {X 0,Y 440.461,Z 320.394,A -85,B 0,C 180,E1 -9986.637,E2 -9986.637} C_VEL
LIN {X 0,Y 434.962,Z 339.48,A -85,B 0,C 180,E1 -9986.599,E2 -9986.599} C_VEL
LIN {X 0,Y 434.396,Z 345.325,A -85,B 0,C 180,E1 -9986.668,E2 -9986.668} C_VEL
LIN {X 0,Y 432.867,Z 416.792,A -85,B 0,C 180,E1 -9987.935,E2 -9987.935} C_VEL
LIN {X 0,Y 432.109,Z 433.658,A -85,B 0,C 180,E1 -9988.427,E2 -9988.427} C_VEL
LIN {X 0,Y 431.045,Z 449.4,A -85,B 0,C 180,E1 -9989.066,E2 -9989.066} C_VEL
LIN {X 0,Y 429.905,Z 464.807,A -85,B 0,C 180,E1 -9989.883,E2 -9989.883} C_VEL
LIN {X 0,Y 428.598,Z 479.006,A -85,B 0,C 180,E1 -9990.806,E2 -9990.806} C_VEL
LIN {X 0,Y 426.994,Z 494.071,A -85,B 0,C 180,E1 -9992.004,E2 -9992.004} C_VEL
LIN {X 0,Y 425.435,Z 507.673,A -85,B 0,C 180,E1 -9993.314,E2 -9993.314} C_VEL
LIN {X 0,Y 423.93,Z 520.295,A -85,B 0,C 180,E1 -9994.754,E2 -9994.754} C_VEL
LIN {X 0,Y 422.598,Z 531.228,A -85,B 0,C 180,E1 -9996.205,E2 -9996.205} C_VEL
LIN {X 0,Y 421.22,Z 542.156,A -85,B 0,C 180,E1 -9997.911,E2 -9997.911} C_VEL
LIN {X 0,Y 420.097,Z 551.51,A -85,B 0,C 180,E1 -9999.63,E2 -9999.63} C_VEL
LIN {X 0,Y 419.103,Z 560.639,A -85,B 0,C 180,E1 -10001.608,E2 -10001.608} C_VEL
LIN {X 0,Y 418.351,Z 568.321,A -85,B 0,C 180,E1 -10003.602,E2 -10003.602} C_VEL
LIN {X 0,Y 417.633,Z 575.765,A -85,B 0,C 180,E1 -10006.015,E2 -10006.015} C_VEL
LIN {X 0,Y 417.327,Z 580.842,A -85,B 0,C 180,E1 -10008.152,E2 -10008.152} C_VEL
LIN {X 0,Y 417.109,Z 583.753,A -85,B 0,C 180,E1 -10009.693,E2 -10009.693} C_VEL
LIN {X 0,Y 416.897,Z 586.846,A -85,B 0,C 180,E1 -10012.001,E2 -10012.001} C_VEL
LIN {X 0,Y 416.804,Z 588.614,A -85,B 0,C 180,E1 -10014.422,E2 -10014.422} C_VEL
LIN {X 0,Y 416.805,Z 588.923,A -85,B 0,C 180,E1 -10016.663,E2 -10016.663} C_VEL
LIN {X 0,Y 416.858,Z 588.109,A -85,B 0,C 180,E1 -10018.755,E2 -10018.755} C_VEL
LIN {X 0,Y 416.984,Z 586.241,A -85,B 0,C 180,E1 -10020.732,E2 -10020.732} C_VEL
LIN {X 0,Y 417.221,Z 582.526,A -85,B 0,C 180,E1 -10023.192,E2 -10023.192} C_VEL
LIN {X 0,Y 417.643,Z 577.556,A -85,B 0,C 180,E1 -10025.489,E2 -10025.489} C_VEL
LIN {X 0,Y 418.131,Z 570.957,A -85,B 0,C 180,E1 -10027.816,E2 -10027.816} C_VEL
LIN {X 0,Y 418.891,Z 563.487,A -85,B 0,C 180,E1 -10029.921,E2 -10029.921} C_VEL
LIN {X 0,Y 419.898,Z 554.364,A -85,B 0,C 180,E1 -10032.027,E2 -10032.027} C_VEL
LIN {X 0,Y 421.282,Z 543.093,A -85,B 0,C 180,E1 -10034.165,E2 -10034.165} C_VEL
LIN {X 0,Y 422.797,Z 531.675,A -85,B 0,C 180,E1 -10035.964,E2 -10035.964} C_VEL
LIN {X 0,Y 424.351,Z 519.462,A -85,B 0,C 180,E1 -10037.586,E2 -10037.586} C_VEL
LIN {X 0,Y 425.787,Z 507.56,A -85,B 0,C 180,E1 -10038.935,E2 -10038.935} C_VEL
LIN {X 0,Y 427.45,Z 493.746,A -85,B 0,C 180,E1 -10040.26,E2 -10040.26} C_VEL
LIN {X 0,Y 428.969,Z 479.648,A -85,B 0,C 180,E1 -10041.388,E2 -10041.388} C_VEL
LIN {X 0,Y 430.405,Z 464.644,A -85,B 0,C 180,E1 -10042.366,E2 -10042.366} C_VEL
LIN {X 0,Y 431.53,Z 450.171,A -85,B 0,C 180,E1 -10043.134,E2 -10043.134} C_VEL
LIN {X 0,Y 432.602,Z 433.977,A -85,B 0,C 180,E1 -10043.799,E2 -10043.799} C_VEL
LIN {X 0,Y 433.473,Z 416.933,A -85,B 0,C 180,E1 -10044.291,E2 -10044.291} C_VEL
LIN {X 0,Y 437.422,Z 245.032,A -85,B 0,C 180,E1 -10047.334,E2 -10047.334} C_VEL
LIN {X 0,Y 429.665,Z 228.976,A -85,B 0,C 180,E1 -10048.326,E2 -10048.326} C_VEL
LIN {X 0,Y 421.466,Z 213.922,A -85,B 0,C 180,E1 -10049.395,E2 -10049.395} C_VEL
LIN {X 0,Y 420.059,Z 211.164,A -85,B 0,C 180,E1 -10049.595,E2 -10049.595} C_VEL
LIN {X 0,Y 418.235,Z 205.7,A -85,B 0,C 180,E1 -10050.629,E2 -10050.629} C_VEL
LIN {X 0,Y 418.223,Z 205.703,A -85,B 0,C 180,E1 -10054.093,E2 -10054.093} C_VEL
LIN {X 0,Y 418.221,Z 205.699,A -85,B 0,C 180,E1 -10057.263,E2 -10057.263} C_VEL
LIN {X 0,Y 418.276,Z 205.693,A -85,B 0,C 180,E1 -10060.364,E2 -10060.364} C_VEL
LIN {X 0,Y 418.31,Z 205.688,A -85,B 0,C 180,E1 -10063.404,E2 -10063.404} C_VEL
LIN {X 0,Y 418.34,Z 205.682,A -85,B 0,C 180,E1 -10066.999,E2 -10066.999} C_VEL
LIN {X 0,Y 418.332,Z 205.691,A -85,B 0,C 180,E1 -10070.328,E2 -10070.328} C_VEL
LIN {X 0,Y 418.464,Z 205.668,A -85,B 0,C 180,E1 -10073.249,E2 -10073.249} C_VEL
LIN {X 0,Y 418.329,Z 205.685,A -85,B 0,C 180,E1 -10075.181,E2 -10075.181} C_VEL
LIN {X 0,Y 418.536,Z 205.662,A -85,B 0,C 180,E1 -10078.075,E2 -10078.075} C_VEL
LIN {X 0,Y 418.665,Z 205.648,A -85,B 0,C 180,E1 -10080,E2 -10080} C_VEL
LIN {X 0,Y 418.494,Z 205.663,A -85,B 0,C 180,E1 -10082.888,E2 -10082.888} C_VEL
LIN {X 0,Y 418.486,Z 205.669,A -85,B 0,C 180,E1 -10086.751,E2 -10086.751} C_VEL
LIN {X 0,Y 418.335,Z 205.688,A -85,B 0,C 180,E1 -10089.671,E2 -10089.671} C_VEL
LIN {X 0,Y 418.34,Z 205.685,A -85,B 0,C 180,E1 -10093.001,E2 -10093.001} C_VEL
LIN {X 0,Y 418.307,Z 205.688,A -85,B 0,C 180,E1 -10096.736,E2 -10096.736} C_VEL
LIN {X 0,Y 418.265,Z 205.697,A -85,B 0,C 180,E1 -10099.791,E2 -10099.791} C_VEL
LIN {X 0,Y 418.232,Z 205.699,A -85,B 0,C 180,E1 -10102.736,E2 -10102.736} C_VEL
LIN {X 0,Y 418.266,Z 205.696,A -85,B 0,C 180,E1 -10105.904,E2 -10105.904} C_VEL
LIN {X 0,Y 418.259,Z 205.696,A -85,B 0,C 180,E1 -10109.162,E2 -10109.162} C_VEL
LIN {X 0,Y 418.252,Z 205.7,A -85,B 0,C 180,E1 -10112.844,E2 -10112.844} C_VEL
LIN {X 0,Y 418.239,Z 205.702,A -85,B 0,C 180,E1 -10116.238,E2 -10116.238} C_VEL
LIN {X 0,Y 418.246,Z 205.702,A -85,B 0,C 180,E1 -10119.682,E2 -10119.682} C_VEL
LIN {X 0,Y 418.224,Z 205.705,A -85,B 0,C 180,E1 -10122.322,E2 -10122.322} C_VEL
LIN {X 0,Y 418.231,Z 205.707,A -85,B 0,C 180,E1 -10125.109,E2 -10125.109} C_VEL
LIN {X 0,Y 418.235,Z 205.705,A -85,B 0,C 180,E1 -10127.767,E2 -10127.767} C_VEL
LIN {X 0,Y 418.248,Z 205.7,A -85,B 0,C 180,E1 -10130.62,E2 -10130.62} C_VEL
LIN {X 0,Y 418.234,Z 205.77,A -85,B 0,C 180,E1 -10132.997,E2 -10132.997} C_VEL
LIN {X 0,Y 423.631,Z 221.449,A -85,B 0,C 180,E1 -10135.664,E2 -10135.664} C_VEL
LIN {X 0,Y 426.438,Z 230.428,A -85,B 0,C 180,E1 -10137.051,E2 -10137.051} C_VEL
